LIN {X 0,Y 272.161,Z 198.873,A -85,B 0,C 180,E1 -18848.578,E2 -18848.578} C_VEL
LIN {X 0,Y 269.803,Z 194.303,A -85,B 0,C 180,E1 -18849.734,E2 -18849.734} C_VEL
LIN {X 0,Y 266.598,Z 188.645,A -85,B 0,C 180,E1 -18851.406,E2 -18851.406} C_VEL
LIN {X 0,Y 262.771,Z 182.274,A -85,B 0,C 180,E1 -18853.688,E2 -18853.688} C_VEL
LIN {X 0,Y 258.268,Z 175.293,A -85,B 0,C 180,E1 -18857.039,E2 -18857.039} C_VEL
LIN {X 0,Y 254.053,Z 169.261,A -85,B 0,C 180,E1 -18861.694,E2 -18861.694} C_VEL
LIN {X 0,Y 252.896,Z 167.097,A -85,B 0,C 180,E1 -18864.05,E2 -18864.05} C_VEL
LIN {X 0,Y 252.189,Z 165.744,A -85,B 0,C 180,E1 -18867.234,E2 -18867.234} C_VEL
LIN {X 0,Y 252.626,Z 165.739,A -85,B 0,C 180,E1 -18870.81,E2 -18870.81} C_VEL
LIN {X 0,Y 254.505,Z 167.542,A -85,B 0,C 180,E1 -18874.522,E2 -18874.522} C_VEL
LIN {X 0,Y 256.623,Z 169.192,A -85,B 0,C 180,E1 -18876.922,E2 -18876.922} C_VEL
LIN {X 0,Y 261.122,Z 174.199,A -85,B 0,C 180,E1 -18880.646,E2 -18880.646} C_VEL
LIN {X 0,Y 265.231,Z 179.251,A -85,B 0,C 180,E1 -18883.234,E2 -18883.234} C_VEL
LIN {X 0,Y 268.61,Z 183.835,A -85,B 0,C 180,E1 -18885.072,E2 -18885.072} C_VEL
LIN {X 0,Y 271.817,Z 188.374,A -85,B 0,C 180,E1 -18886.589,E2 -18886.589} C_VEL
LIN {X 0,Y 276.316,Z 195.238,A -85,B 0,C 180,E1 -18888.534,E2 -18888.534} C_VEL
LIN {X 0,Y 282.169,Z 206.406,A -85,B 0,C 180,E1 -18890.864,E2 -18890.864} C_VEL
LIN {X 0,Y 283.422,Z 209.263,A -85,B 0,C 180,E1 -18891.341,E2 -18891.341} C_VEL
LIN {X 0,Y 278.255,Z 265.436,A -85,B 0,C 180,E1 -18893.382,E2 -18893.382} C_VEL
LIN {X 0,Y 276.562,Z 278.897,A -85,B 0,C 180,E1 -18894.165,E2 -18894.165} C_VEL
LIN {X 0,Y 274.571,Z 290.757,A -85,B 0,C 180,E1 -18895.117,E2 -18895.117} C_VEL
LIN {X 0,Y 271.722,Z 303.647,A -85,B 0,C 180,E1 -18896.478,E2 -18896.478} C_VEL
LIN {X 0,Y 268.861,Z 314.419,A -85,B 0,C 180,E1 -18897.94,E2 -18897.94} C_VEL
LIN {X 0,Y 265.559,Z 325.122,A -85,B 0,C 180,E1 -18899.802,E2 -18899.802} C_VEL
LIN {X 0,Y 262.251,Z 334.733,A -85,B 0,C 180,E1 -18901.909,E2 -18901.909} C_VEL
LIN {X 0,Y 258.95,Z 343.17,A -85,B 0,C 180,E1 -18904.279,E2 -18904.279} C_VEL
LIN {X 0,Y 255.863,Z 350.386,A -85,B 0,C 180,E1 -18906.908,E2 -18906.908} C_VEL
LIN {X 0,Y 253.246,Z 355.852,A -85,B 0,C 180,E1 -18909.584,E2 -18909.584} C_VEL
LIN {X 0,Y 251.415,Z 359.437,A -85,B 0,C 180,E1 -18911.933,E2 -18911.933} C_VEL
LIN {X 0,Y 249.746,Z 362.315,A -85,B 0,C 180,E1 -18914.67,E2 -18914.67} C_VEL
LIN {X 0,Y 248.899,Z 363.505,A -85,B 0,C 180,E1 -18916.401,E2 -18916.401} C_VEL
LIN {X 0,Y 248.206,Z 364.182,A -85,B 0,C 180,E1 -18918.147,E2 -18918.147} C_VEL
LIN {X 0,Y 247.543,Z 364.385,A -85,B 0,C 180,E1 -18920.461,E2 -18920.461} C_VEL
LIN {X 0,Y 247.05,Z 363.363,A -85,B 0,C 180,E1 -18923.469,E2 -18923.469} C_VEL
LIN {X 0,Y 246.899,Z 362.091,A -85,B 0,C 180,E1 -18925.275,E2 -18925.275} C_VEL
LIN {X 0,Y 247.04,Z 358.996,A -85,B 0,C 180,E1 -18928.125,E2 -18928.125} C_VEL
LIN {X 0,Y 247.409,Z 354.863,A -85,B 0,C 180,E1 -18930.751,E2 -18930.751} C_VEL
LIN {X 0,Y 247.931,Z 348.96,A -85,B 0,C 180,E1 -18933.556,E2 -18933.556} C_VEL
LIN {X 0,Y 248.602,Z 342.47,A -85,B 0,C 180,E1 -18935.968,E2 -18935.968} C_VEL
LIN {X 0,Y 249.5,Z 334.669,A -85,B 0,C 180,E1 -18938.294,E2 -18938.294} C_VEL
LIN {X 0,Y 250.624,Z 325.418,A -85,B 0,C 180,E1 -18940.519,E2 -18940.519} C_VEL
LIN {X 0,Y 251.866,Z 314.797,A -85,B 0,C 180,E1 -18942.583,E2 -18942.583} C_VEL
LIN {X 0,Y 253.111,Z 304.125,A -85,B 0,C 180,E1 -18944.236,E2 -18944.236} C_VEL
LIN {X 0,Y 254.279,Z 291.49,A -85,B 0,C 180,E1 -18945.797,E2 -18945.797} C_VEL
LIN {X 0,Y 255.46,Z 277.915,A -85,B 0,C 180,E1 -18947.043,E2 -18947.043} C_VEL
LIN {X 0,Y 256.185,Z 264.7,A -85,B 0,C 180,E1 -18947.927,E2 -18947.927} C_VEL
LIN {X 0,Y 256.929,Z 247.419,A -85,B 0,C 180,E1 -18948.64,E2 -18948.64} C_VEL
LIN {X 0,Y 259.313,Z 186.757,A -85,B 0,C 180,E1 -18950.805,E2 -18950.805} C_VEL
LIN {X 0,Y 254.059,Z 171.401,A -85,B 0,C 180,E1 -18951.759,E2 -18951.759} C_VEL
LIN {X 0,Y 249.108,Z 157.454,A -85,B 0,C 180,E1 -18952.7,E2 -18952.7} C_VEL
LIN {X 0,Y 249.056,Z 157.463,A -85,B 0,C 180,E1 -18955.641,E2 -18955.641} C_VEL
LIN {X 0,Y 249.052,Z 157.465,A -85,B 0,C 180,E1 -18959.472,E2 -18959.472} C_VEL
LIN {X 0,Y 249.074,Z 157.462,A -85,B 0,C 180,E1 -18963.162,E2 -18963.162} C_VEL
LIN {X 0,Y 249.078,Z 157.458,A -85,B 0,C 180,E1 -18966.732,E2 -18966.732} C_VEL
LIN {X 0,Y 249.092,Z 157.454,A -85,B 0,C 180,E1 -18970.209,E2 -18970.209} C_VEL
LIN {X 0,Y 249.194,Z 157.443,A -85,B 0,C 180,E1 -18973.618,E2 -18973.618} C_VEL
LIN {X 0,Y 249.25,Z 157.436,A -85,B 0,C 180,E1 -18978.616,E2 -18978.616} C_VEL
LIN {X 0,Y 249.478,Z 157.406,A -85,B 0,C 180,E1 -18981.902,E2 -18981.902} C_VEL
LIN {X 0,Y 249.435,Z 157.414,A -85,B 0,C 180,E1 -18986.769,E2 -18986.769} C_VEL
LIN {X 0,Y 249.727,Z 157.376,A -85,B 0,C 180,E1 -18989.999,E2 -18989.999} C_VEL
LIN {X 0,Y 249.434,Z 157.412,A -85,B 0,C 180,E1 -18993.23,E2 -18993.23} C_VEL
LIN {X 0,Y 249.478,Z 157.408,A -85,B 0,C 180,E1 -18998.097,E2 -18998.097} C_VEL
LIN {X 0,Y 249.251,Z 157.433,A -85,B 0,C 180,E1 -19001.383,E2 -19001.383} C_VEL
LIN {X 0,Y 249.24,Z 157.44,A -85,B 0,C 180,E1 -19006.378,E2 -19006.378} C_VEL
LIN {X 0,Y 249.081,Z 157.455,A -85,B 0,C 180,E1 -19011.518,E2 -19011.518} C_VEL
LIN {X 0,Y 249.115,Z 157.452,A -85,B 0,C 180,E1 -19015.475,E2 -19015.475} C_VEL
LIN {X 0,Y 249.084,Z 157.455,A -85,B 0,C 180,E1 -19018.994,E2 -19018.994} C_VEL
LIN {X 0,Y 249.033,Z 157.464,A -85,B 0,C 180,E1 -19022.425,E2 -19022.425} C_VEL
LIN {X 0,Y 249.072,Z 157.458,A -85,B 0,C 180,E1 -19026.337,E2 -19026.337} C_VEL
LIN {X 0,Y 249.074,Z 157.458,A -85,B 0,C 180,E1 -19030.464,E2 -19030.464} C_VEL
LIN {X 0,Y 249.019,Z 157.462,A -85,B 0,C 180,E1 -19034.875,E2 -19034.875} C_VEL
LIN {X 0,Y 249.049,Z 157.461,A -85,B 0,C 180,E1 -19037.371,E2 -19037.371} C_VEL
LIN {X 0,Y 249.048,Z 157.463,A -85,B 0,C 180,E1 -19041.624,E2 -19041.624} C_VEL
LIN {X 0,Y 249.059,Z 157.463,A -85,B 0,C 180,E1 -19045.643,E2 -19045.643} C_VEL
LIN {X 0,Y 249.049,Z 157.463,A -85,B 0,C 180,E1 -19049.473,E2 -19049.473} C_VEL
LIN {X 0,Y 249.072,Z 157.459,A -85,B 0,C 180,E1 -19053.163,E2 -19053.163} C_VEL
LIN {X 0,Y 249.077,Z 157.457,A -85,B 0,C 180,E1 -19056.733,E2 -19056.733} C_VEL
LIN {X 0,Y 249.108,Z 157.451,A -85,B 0,C 180,E1 -19060.212,E2 -19060.212} C_VEL
LIN {X 0,Y 249.239,Z 157.438,A -85,B 0,C 180,E1 -19063.622,E2 -19063.622} C_VEL
LIN {X 0,Y 249.251,Z 157.434,A -85,B 0,C 180,E1 -19068.617,E2 -19068.617} C_VEL
LIN {X 0,Y 249.477,Z 157.407,A -85,B 0,C 180,E1 -19071.903,E2 -19071.903} C_VEL
LIN {X 0,Y 249.434,Z 157.413,A -85,B 0,C 180,E1 -19076.77,E2 -19076.77} C_VEL
LIN {X 0,Y 249.727,Z 157.376,A -85,B 0,C 180,E1 -19080.001,E2 -19080.001} C_VEL
LIN {X 0,Y 249.435,Z 157.411,A -85,B 0,C 180,E1 -19083.231,E2 -19083.231} C_VEL
LIN {X 0,Y 249.483,Z 157.407,A -85,B 0,C 180,E1 -19088.098,E2 -19088.098} C_VEL
LIN {X 0,Y 249.252,Z 157.433,A -85,B 0,C 180,E1 -19091.384,E2 -19091.384} C_VEL
LIN {X 0,Y 249.206,Z 157.441,A -85,B 0,C 180,E1 -19095.849,E2 -19095.849} C_VEL
LIN {X 0,Y 248.917,Z 157.479,A -85,B 0,C 180,E1 -19096.751,E2 -19096.751} C_VEL
LIN {X 0,Y 247.56,Z 157.65,A -85,B 0,C 180,E1 -19098.081,E2 -19098.081} C_VEL
LIN {X 0,Y 243.133,Z 158.197,A -85,B 0,C 180,E1 -19101.182,E2 -19101.182} C_VEL
LIN {X 0,Y 242.07,Z 158.332,A -85,B 0,C 180,E1 -19102.572,E2 -19102.572} C_VEL
LIN {X 0,Y 241.992,Z 158.337,A -85,B 0,C 180,E1 -19103.044,E2 -19103.044} C_VEL
LIN {X 0,Y 242.066,Z 158.331,A -85,B 0,C 180,E1 -19105.839,E2 -19105.839} C_VEL
LIN {X 0,Y 242.03,Z 158.333,A -85,B 0,C 180,E1 -19109.581,E2 -19109.581} C_VEL
LIN {X 0,Y 241.991,Z 158.34,A -85,B 0,C 180,E1 -19113.492,E2 -19113.492} C_VEL
LIN {X 0,Y 242.011,Z 158.335,A -85,B 0,C 180,E1 -19117.579,E2 -19117.579} C_VEL
LIN {X 0,Y 241.954,Z 158.348,A -85,B 0,C 180,E1 -19121.92,E2 -19121.92} C_VEL
LIN {X 0,Y 241.935,Z 158.347,A -85,B 0,C 180,E1 -19126.572,E2 -19126.572} C_VEL
LIN {X 0,Y 241.957,Z 158.345,A -85,B 0,C 180,E1 -19130.282,E2 -19130.282} C_VEL
LIN {X 0,Y 242.087,Z 158.358,A -85,B 0,C 180,E1 -19134.698,E2 -19134.698} C_VEL
LIN {X 0,Y 244.791,Z 171.849,A -85,B 0,C 180,E1 -19139.464,E2 -19139.464} C_VEL
LIN {X 0,Y 246.244,Z 179.046,A -85,B 0,C 180,E1 -19141.867,E2 -19141.867} C_VEL
LIN {X 0,Y 251.436,Z 230.762,A -85,B 0,C 180,E1 -19144.295,E2 -19144.295} C_VEL
LIN {X 0,Y 249.178,Z 289.171,A -85,B 0,C 180,E1 -19146.523,E2 -19146.523} C_VEL
LIN {X 0,Y 248.278,Z 301.999,A -85,B 0,C 180,E1 -19147.315,E2 -19147.315} C_VEL
LIN {X 0,Y 247.106,Z 313.577,A -85,B 0,C 180,E1 -19148.301,E2 -19148.301} C_VEL
LIN {X 0,Y 245.772,Z 325.986,A -85,B 0,C 180,E1 -19149.714,E2 -19149.714} C_VEL
LIN {X 0,Y 244.389,Z 337.207,A -85,B 0,C 180,E1 -19151.342,E2 -19151.342} C_VEL
LIN {X 0,Y 243.042,Z 347.408,A -85,B 0,C 180,E1 -19153.193,E2 -19153.193} C_VEL
LIN {X 0,Y 242.034,Z 356.689,A -85,B 0,C 180,E1 -19155.282,E2 -19155.282} C_VEL
LIN {X 0,Y 241.063,Z 365.717,A -85,B 0,C 180,E1 -19157.798,E2 -19157.798} C_VEL
LIN {X 0,Y 240.491,Z 372.88,A -85,B 0,C 180,E1 -19160.327,E2 -19160.327} C_VEL
LIN {X 0,Y 240.242,Z 379.387,A -85,B 0,C 180,E1 -19163.281,E2 -19163.281} C_VEL
LIN {X 0,Y 240.242,Z 383.565,A -85,B 0,C 180,E1 -19165.807,E2 -19165.807} C_VEL
LIN {X 0,Y 240.167,Z 386.556,A -85,B 0,C 180,E1 -19168.324,E2 -19168.324} C_VEL
LIN {X 0,Y 240.34,Z 387.982,A -85,B 0,C 180,E1 -19170.001,E2 -19170.001} C_VEL
LIN {X 0,Y 240.01,Z 389.407,A -85,B 0,C 180,E1 -19173.358,E2 -19173.358} C_VEL
LIN {X 0,Y 239.853,Z 389.5,A -85,B 0,C 180,E1 -19175.044,E2 -19175.044} C_VEL
LIN {X 0,Y 239.896,Z 389.18,A -85,B 0,C 180,E1 -19176.73,E2 -19176.73} C_VEL
LIN {X 0,Y 240.5,Z 387.299,A -85,B 0,C 180,E1 -19180.099,E2 -19180.099} C_VEL
LIN {X 0,Y 241.037,Z 385.763,A -85,B 0,C 180,E1 -19181.778,E2 -19181.778} C_VEL
LIN {X 0,Y 242.247,Z 382.634,A -85,B 0,C 180,E1 -19184.277,E2 -19184.277} C_VEL
LIN {X 0,Y 244.074,Z 378.522,A -85,B 0,C 180,E1 -19186.736,E2 -19186.736} C_VEL
LIN {X 0,Y 246.158,Z 373.316,A -85,B 0,C 180,E1 -19189.168,E2 -19189.168} C_VEL
LIN {X 0,Y 248.789,Z 366.863,A -85,B 0,C 180,E1 -19191.546,E2 -19191.546} C_VEL
LIN {X 0,Y 252.077,Z 358.919,A -85,B 0,C 180,E1 -19193.846,E2 -19193.846} C_VEL
LIN {X 0,Y 255.101,Z 350.996,A -85,B 0,C 180,E1 -19195.717,E2 -19195.717} C_VEL
LIN {X 0,Y 258.965,Z 340.381,A -85,B 0,C 180,E1 -19197.695,E2 -19197.695} C_VEL
LIN {X 0,Y 262.272,Z 329.818,A -85,B 0,C 180,E1 -19199.278,E2 -19199.278} C_VEL
LIN {X 0,Y 265.545,Z 318.133,A -85,B 0,C 180,E1 -19200.63,E2 -19200.63} C_VEL
LIN {X 0,Y 268.928,Z 304.154,A -85,B 0,C 180,E1 -19201.842,E2 -19201.842} C_VEL
LIN {X 0,Y 271.411,Z 290.859,A -85,B 0,C 180,E1 -19202.666,E2 -19202.666} C_VEL
LIN {X 0,Y 273.13,Z 276.909,A -85,B 0,C 180,E1 -19203.288,E2 -19203.288} C_VEL
LIN {X 0,Y 276.662,Z 237.361,A -85,B 0,C 180,E1 -19204.745,E2 -19204.745} C_VEL
LIN {X 0,Y 275.715,Z 223.84,A -85,B 0,C 180,E1 -19205.824,E2 -19205.824} C_VEL
LIN {X 0,Y 275.099,Z 218.549,A -85,B 0,C 180,E1 -19206.339,E2 -19206.339} C_VEL
LIN {X 0,Y 271.495,Z 209.724,A -85,B 0,C 180,E1 -19208.005,E2 -19208.005} C_VEL
LIN {X 0,Y 267.297,Z 200.762,A -85,B 0,C 180,E1 -19210.135,E2 -19210.135} C_VEL
LIN {X 0,Y 263.888,Z 194.57,A -85,B 0,C 180,E1 -19212.024,E2 -19212.024} C_VEL
LIN {X 0,Y 260.503,Z 188.645,A -85,B 0,C 180,E1 -19214.173,E2 -19214.173} C_VEL
LIN {X 0,Y 256.366,Z 181.862,A -85,B 0,C 180,E1 -19217.45,E2 -19217.45} C_VEL
LIN {X 0,Y 252.367,Z 175.801,A -85,B 0,C 180,E1 -19222.217,E2 -19222.217} C_VEL
LIN {X 0,Y 251.349,Z 173.787,A -85,B 0,C 180,E1 -19224.568,E2 -19224.568} C_VEL
LIN {X 0,Y 250.805,Z 172.582,A -85,B 0,C 180,E1 -19227.831,E2 -19227.831} C_VEL
LIN {X 0,Y 251.371,Z 172.83,A -85,B 0,C 180,E1 -19231.136,E2 -19231.136} C_VEL
LIN {X 0,Y 253.916,Z 175.089,A -85,B 0,C 180,E1 -19235.469,E2 -19235.469} C_VEL
LIN {X 0,Y 255.04,Z 176.102,A -85,B 0,C 180,E1 -19236.744,E2 -19236.744} C_VEL
LIN {X 0,Y 259.027,Z 180.69,A -85,B 0,C 180,E1 -19240.204,E2 -19240.204} C_VEL
LIN {X 0,Y 262.925,Z 185.673,A -85,B 0,C 180,E1 -19242.798,E2 -19242.798} C_VEL
LIN {X 0,Y 266.299,Z 190.371,A -85,B 0,C 180,E1 -19244.697,E2 -19244.697} C_VEL
LIN {X 0,Y 270.776,Z 197.051,A -85,B 0,C 180,E1 -19246.892,E2 -19246.892} C_VEL
LIN {X 0,Y 274.226,Z 203.049,A -85,B 0,C 180,E1 -19248.441,E2 -19248.441} C_VEL
LIN {X 0,Y 278.658,Z 212.019,A -85,B 0,C 180,E1 -19250.306,E2 -19250.306} C_VEL
LIN {X 0,Y 273.522,Z 265.759,A -85,B 0,C 180,E1 -19252.285,E2 -19252.285} C_VEL
LIN {X 0,Y 271.809,Z 278.655,A -85,B 0,C 180,E1 -19253.038,E2 -19253.038} C_VEL
LIN {X 0,Y 269.661,Z 290.779,A -85,B 0,C 180,E1 -19254.016,E2 -19254.016} C_VEL
LIN {X 0,Y 266.869,Z 302.828,A -85,B 0,C 180,E1 -19255.289,E2 -19255.289} C_VEL
LIN {X 0,Y 263.827,Z 313.801,A -85,B 0,C 180,E1 -19256.754,E2 -19256.754} C_VEL
LIN {X 0,Y 260.656,Z 323.839,A -85,B 0,C 180,E1 -19258.454,E2 -19258.454} C_VEL
LIN {X 0,Y 257.324,Z 332.949,A -85,B 0,C 180,E1 -19260.391,E2 -19260.391} C_VEL
LIN {X 0,Y 253.79,Z 341.769,A -85,B 0,C 180,E1 -19262.776,E2 -19262.776} C_VEL
LIN {X 0,Y 250.61,Z 348.832,A -85,B 0,C 180,E1 -19265.229,E2 -19265.229} C_VEL
LIN {X 0,Y 248.095,Z 353.926,A -85,B 0,C 180,E1 -19267.484,E2 -19267.484} C_VEL
LIN {X 0,Y 245.868,Z 358.084,A -85,B 0,C 180,E1 -19269.875,E2 -19269.875} C_VEL
LIN {X 0,Y 244.28,Z 360.854,A -85,B 0,C 180,E1 -19271.986,E2 -19271.986} C_VEL
LIN {X 0,Y 242.399,Z 363.55,A -85,B 0,C 180,E1 -19275.125,E2 -19275.125} C_VEL
LIN {X 0,Y 241.591,Z 364.425,A -85,B 0,C 180,E1 -19276.911,E2 -19276.911} C_VEL
LIN {X 0,Y 240.912,Z 364.831,A -85,B 0,C 180,E1 -19278.717,E2 -19278.717} C_VEL
LIN {X 0,Y 240.405,Z 364.695,A -85,B 0,C 180,E1 -19280.692,E2 -19280.692} C_VEL
LIN {X 0,Y 240.068,Z 364.163,A -85,B 0,C 180,E1 -19282.369,E2 -19282.369} C_VEL
LIN {X 0,Y 239.846,Z 362.691,A -85,B 0,C 180,E1 -19284.718,E2 -19284.718} C_VEL
LIN {X 0,Y 239.915,Z 359.335,A -85,B 0,C 180,E1 -19287.949,E2 -19287.949} C_VEL
LIN {X 0,Y 240.306,Z 354.927,A -85,B 0,C 180,E1 -19290.783,E2 -19290.783} C_VEL
LIN {X 0,Y 240.873,Z 348.928,A -85,B 0,C 180,E1 -19293.666,E2 -19293.666} C_VEL
LIN {X 0,Y 241.548,Z 342.465,A -85,B 0,C 180,E1 -19296.099,E2 -19296.099} C_VEL
LIN {X 0,Y 242.477,Z 334.497,A -85,B 0,C 180,E1 -19298.502,E2 -19298.502} C_VEL
LIN {X 0,Y 243.618,Z 325.33,A -85,B 0,C 180,E1 -19300.744,E2 -19300.744} C_VEL
LIN {X 0,Y 244.706,Z 315.837,A -85,B 0,C 180,E1 -19302.643,E2 -19302.643} C_VEL
LIN {X 0,Y 246.029,Z 304.743,A -85,B 0,C 180,E1 -19304.426,E2 -19304.426} C_VEL
LIN {X 0,Y 247.246,Z 292.317,A -85,B 0,C 180,E1 -19306.013,E2 -19306.013} C_VEL
LIN {X 0,Y 248.356,Z 279.879,A -85,B 0,C 180,E1 -19307.222,E2 -19307.222} C_VEL
LIN {X 0,Y 249.236,Z 265.509,A -85,B 0,C 180,E1 -19308.238,E2 -19308.238} C_VEL
LIN {X 0,Y 249.988,Z 249.032,A -85,B 0,C 180,E1 -19308.957,E2 -19308.957} C_VEL
LIN {X 0,Y 252.492,Z 188.132,A -85,B 0,C 180,E1 -19311.209,E2 -19311.209} C_VEL
LIN {X 0,Y 245.433,Z 167.869,A -85,B 0,C 180,E1 -19312.519,E2 -19312.519} C_VEL
LIN {X 0,Y 242.051,Z 158.335,A -85,B 0,C 180,E1 -19313.182,E2 -19313.182} C_VEL
LIN {X 0,Y 241.993,Z 158.343,A -85,B 0,C 180,E1 -19317.374,E2 -19317.374} C_VEL
LIN {X 0,Y 242.037,Z 158.336,A -85,B 0,C 180,E1 -19320.586,E2 -19320.586} C_VEL
LIN {X 0,Y 242.067,Z 158.331,A -85,B 0,C 180,E1 -19324.182,E2 -19324.182} C_VEL
LIN {X 0,Y 242.051,Z 158.332,A -85,B 0,C 180,E1 -19328.297,E2 -19328.297} C_VEL
LIN {X 0,Y 242.114,Z 158.327,A -85,B 0,C 180,E1 -19333.315,E2 -19333.315} C_VEL
LIN {X 0,Y 242.182,Z 158.315,A -85,B 0,C 180,E1 -19338.279,E2 -19338.279} C_VEL
LIN {X 0,Y 242.425,Z 158.286,A -85,B 0,C 180,E1 -19341.665,E2 -19341.665} C_VEL
LIN {X 0,Y 242.258,Z 158.308,A -85,B 0,C 180,E1 -19345.007,E2 -19345.007} C_VEL
LIN {X 0,Y 242.635,Z 158.26,A -85,B 0,C 180,E1 -19348.34,E2 -19348.34} C_VEL
LIN {X 0,Y 242.635,Z 158.258,A -85,B 0,C 180,E1 -19351.659,E2 -19351.659} C_VEL
LIN {X 0,Y 242.43,Z 158.289,A -85,B 0,C 180,E1 -19356.658,E2 -19356.658} C_VEL
LIN {X 0,Y 242.312,Z 158.299,A -85,B 0,C 180,E1 -19360.021,E2 -19360.021} C_VEL
LIN {X 0,Y 242.165,Z 158.318,A -85,B 0,C 180,E1 -19365.14,E2 -19365.14} C_VEL
LIN {X 0,Y 242.07,Z 158.33,A -85,B 0,C 180,E1 -19368.624,E2 -19368.624} C_VEL
LIN {X 0,Y 242.004,Z 158.34,A -85,B 0,C 180,E1 -19372.18,E2 -19372.18} C_VEL
LIN {X 0,Y 242.064,Z 158.331,A -85,B 0,C 180,E1 -19375.838,E2 -19375.838} C_VEL
LIN {X 0,Y 242.029,Z 158.334,A -85,B 0,C 180,E1 -19379.58,E2 -19379.58} C_VEL
LIN {X 0,Y 241.989,Z 158.34,A -85,B 0,C 180,E1 -19383.491,E2 -19383.491} C_VEL
LIN {X 0,Y 242.01,Z 158.337,A -85,B 0,C 180,E1 -19387.577,E2 -19387.577} C_VEL
LIN {X 0,Y 241.982,Z 158.344,A -85,B 0,C 180,E1 -19391.912,E2 -19391.912} C_VEL
LIN {X 0,Y 241.982,Z 158.34,A -85,B 0,C 180,E1 -19396.558,E2 -19396.558} C_VEL
LIN {X 0,Y 241.985,Z 158.34,A -85,B 0,C 180,E1 -19400.287,E2 -19400.287} C_VEL
LIN {X 0,Y 242.033,Z 158.333,A -85,B 0,C 180,E1 -19404.498,E2 -19404.498} C_VEL
LIN {X 0,Y 241.973,Z 158.341,A -85,B 0,C 180,E1 -19408.48,E2 -19408.48} C_VEL
LIN {X 0,Y 242.006,Z 158.336,A -85,B 0,C 180,E1 -19412.313,E2 -19412.313} C_VEL
LIN {X 0,Y 242.055,Z 158.332,A -85,B 0,C 180,E1 -19416.016,E2 -19416.016} C_VEL
LIN {X 0,Y 242.035,Z 158.335,A -85,B 0,C 180,E1 -19419.608,E2 -19419.608} C_VEL
LIN {X 0,Y 242.161,Z 158.322,A -85,B 0,C 180,E1 -19423.279,E2 -19423.279} C_VEL
LIN {X 0,Y 242.184,Z 158.313,A -85,B 0,C 180,E1 -19428.28,E2 -19428.28} C_VEL
LIN {X 0,Y 242.424,Z 158.286,A -85,B 0,C 180,E1 -19431.666,E2 -19431.666} C_VEL
LIN {X 0,Y 242.258,Z 158.308,A -85,B 0,C 180,E1 -19435.008,E2 -19435.008} C_VEL
LIN {X 0,Y 242.635,Z 158.259,A -85,B 0,C 180,E1 -19438.341,E2 -19438.341} C_VEL
LIN {X 0,Y 242.635,Z 158.259,A -85,B 0,C 180,E1 -19441.66,E2 -19441.66} C_VEL
LIN {X 0,Y 242.433,Z 158.287,A -85,B 0,C 180,E1 -19446.659,E2 -19446.659} C_VEL
LIN {X 0,Y 242.344,Z 158.296,A -85,B 0,C 180,E1 -19450.021,E2 -19450.021} C_VEL
LIN {X 0,Y 242.166,Z 158.318,A -85,B 0,C 180,E1 -19455.141,E2 -19455.141} C_VEL
LIN {X 0,Y 242.072,Z 158.331,A -85,B 0,C 180,E1 -19458.625,E2 -19458.625} C_VEL
LIN {X 0,Y 241.992,Z 158.337,A -85,B 0,C 180,E1 -19463.044,E2 -19463.044} C_VEL
LIN {X 0,Y 241.352,Z 158.423,A -85,B 0,C 180,E1 -19464.432,E2 -19464.432} C_VEL
LIN {X 0,Y 238.523,Z 158.772,A -85,B 0,C 180,E1 -19466.696,E2 -19466.696} C_VEL
LIN {X 0,Y 236.093,Z 159.074,A -85,B 0,C 180,E1 -19468.541,E2 -19468.541} C_VEL
LIN {X 0,Y 235.031,Z 159.206,A -85,B 0,C 180,E1 -19469.972,E2 -19469.972} C_VEL
LIN {X 0,Y 234.935,Z 159.219,A -85,B 0,C 180,E1 -19470.458,E2 -19470.458} C_VEL
LIN {X 0,Y 234.96,Z 159.216,A -85,B 0,C 180,E1 -19474.634,E2 -19474.634} C_VEL
LIN {X 0,Y 234.942,Z 159.217,A -85,B 0,C 180,E1 -19478.945,E2 -19478.945} C_VEL
LIN {X 0,Y 234.921,Z 159.221,A -85,B 0,C 180,E1 -19483.479,E2 -19483.479} C_VEL
LIN {X 0,Y 234.888,Z 159.225,A -85,B 0,C 180,E1 -19486.515,E2 -19486.515} C_VEL
LIN {X 0,Y 234.919,Z 159.221,A -85,B 0,C 180,E1 -19491.08,E2 -19491.08} C_VEL
LIN {X 0,Y 235.058,Z 159.348,A -85,B 0,C 180,E1 -19494.418,E2 -19494.418} C_VEL
LIN {X 0,Y 237.284,Z 170.542,A -85,B 0,C 180,E1 -19498.505,E2 -19498.505} C_VEL
LIN {X 0,Y 238.974,Z 178.656,A -85,B 0,C 180,E1 -19501.322,E2 -19501.322} C_VEL
LIN {X 0,Y 239.927,Z 182.771,A -85,B 0,C 180,E1 -19501.567,E2 -19501.567} C_VEL
LIN {X 0,Y 244.528,Z 231.857,A -85,B 0,C 180,E1 -19503.924,E2 -19503.924} C_VEL
LIN {X 0,Y 242.294,Z 288.298,A -85,B 0,C 180,E1 -19506.155,E2 -19506.155} C_VEL
LIN {X 0,Y 241.354,Z 301.216,A -85,B 0,C 180,E1 -19506.966,E2 -19506.966} C_VEL
LIN {X 0,Y 240.074,Z 313.903,A -85,B 0,C 180,E1 -19508.085,E2 -19508.085} C_VEL
LIN {X 0,Y 238.715,Z 326.148,A -85,B 0,C 180,E1 -19509.537,E2 -19509.537} C_VEL
LIN {X 0,Y 237.253,Z 337.811,A -85,B 0,C 180,E1 -19511.303,E2 -19511.303} C_VEL
LIN {X 0,Y 235.955,Z 347.372,A -85,B 0,C 180,E1 -19513.118,E2 -19513.118} C_VEL
LIN {X 0,Y 234.942,Z 356.6,A -85,B 0,C 180,E1 -19515.271,E2 -19515.271} C_VEL
LIN {X 0,Y 233.976,Z 365.573,A -85,B 0,C 180,E1 -19517.863,E2 -19517.863} C_VEL
LIN {X 0,Y 233.417,Z 372.681,A -85,B 0,C 180,E1 -19520.469,E2 -19520.469} C_VEL
LIN {X 0,Y 233.181,Z 378.316,A -85,B 0,C 180,E1 -19523.076,E2 -19523.076} C_VEL
LIN {X 0,Y 233.188,Z 382.654,A -85,B 0,C 180,E1 -19525.68,E2 -19525.68} C_VEL
LIN {X 0,Y 233.097,Z 385.784,A -85,B 0,C 180,E1 -19528.273,E2 -19528.273} C_VEL
LIN {X 0,Y 233.262,Z 387.301,A -85,B 0,C 180,E1 -19530.001,E2 -19530.001} C_VEL
LIN {X 0,Y 232.969,Z 388.309,A -85,B 0,C 180,E1 -19531.729,E2 -19531.729} C_VEL
LIN {X 0,Y 232.937,Z 388.888,A -85,B 0,C 180,E1 -19533.46,E2 -19533.46} C_VEL
LIN {X 0,Y 232.846,Z 388.825,A -85,B 0,C 180,E1 -19536.935,E2 -19536.935} C_VEL
LIN {X 0,Y 233.084,Z 388.195,A -85,B 0,C 180,E1 -19538.672,E2 -19538.672} C_VEL
LIN {X 0,Y 234.042,Z 385.677,A -85,B 0,C 180,E1 -19542.135,E2 -19542.135} C_VEL
LIN {X 0,Y 235.358,Z 382.732,A -85,B 0,C 180,E1 -19544.704,E2 -19544.704} C_VEL
LIN {X 0,Y 237.278,Z 378.785,A -85,B 0,C 180,E1 -19547.23,E2 -19547.23} C_VEL
LIN {X 0,Y 239.808,Z 372.863,A -85,B 0,C 180,E1 -19550.113,E2 -19550.113} C_VEL
LIN {X 0,Y 242.783,Z 366.383,A -85,B 0,C 180,E1 -19552.555,E2 -19552.555} C_VEL
LIN {X 0,Y 246.306,Z 358.502,A -85,B 0,C 180,E1 -19554.89,E2 -19554.89} C_VEL
LIN {X 0,Y 249.51,Z 350.573,A -85,B 0,C 180,E1 -19556.788,E2 -19556.788} C_VEL
LIN {X 0,Y 253.59,Z 339.938,A -85,B 0,C 180,E1 -19558.786,E2 -19558.786} C_VEL
LIN {X 0,Y 257.104,Z 329.488,A -85,B 0,C 180,E1 -19560.379,E2 -19560.379} C_VEL
LIN {X 0,Y 260.083,Z 319.603,A -85,B 0,C 180,E1 -19561.572,E2 -19561.572} C_VEL
LIN {X 0,Y 263.562,Z 306.217,A -85,B 0,C 180,E1 -19562.796,E2 -19562.796} C_VEL
LIN {X 0,Y 266.265,Z 293.281,A -85,B 0,C 180,E1 -19563.662,E2 -19563.662} C_VEL
LIN {X 0,Y 268.276,Z 279.041,A -85,B 0,C 180,E1 -19564.337,E2 -19564.337} C_VEL
LIN {X 0,Y 272.163,Z 238.757,A -85,B 0,C 180,E1 -19565.854,E2 -19565.854} C_VEL
LIN {X 0,Y 271.147,Z 222.952,A -85,B 0,C 180,E1 -19567.197,E2 -19567.197} C_VEL
LIN {X 0,Y 268.34,Z 215.423,A -85,B 0,C 180,E1 -19568.626,E2 -19568.626} C_VEL
LIN {X 0,Y 264.254,Z 206.386,A -85,B 0,C 180,E1 -19570.815,E2 -19570.815} C_VEL
LIN {X 0,Y 261.112,Z 200.322,A -85,B 0,C 180,E1 -19572.712,E2 -19572.712} C_VEL
LIN {X 0,Y 258.062,Z 194.689,A -85,B 0,C 180,E1 -19574.821,E2 -19574.821} C_VEL
LIN {X 0,Y 254.394,Z 188.377,A -85,B 0,C 180,E1 -19577.936,E2 -19577.936} C_VEL
LIN {X 0,Y 250.788,Z 182.536,A -85,B 0,C 180,E1 -19582.571,E2 -19582.571} C_VEL
LIN {X 0,Y 249.96,Z 180.766,A -85,B 0,C 180,E1 -19584.626,E2 -19584.626} C_VEL
LIN {X 0,Y 249.46,Z 179.574,A -85,B 0,C 180,E1 -19587.693,E2 -19587.693} C_VEL
LIN {X 0,Y 249.948,Z 179.744,A -85,B 0,C 180,E1 -19590.957,E2 -19590.957} C_VEL
LIN {X 0,Y 252.416,Z 181.968,A -85,B 0,C 180,E1 -19595.313,E2 -19595.313} C_VEL
LIN {X 0,Y 253.64,Z 183.312,A -85,B 0,C 180,E1 -19596.77,E2 -19596.77} C_VEL
LIN {X 0,Y 257.047,Z 187.313,A -85,B 0,C 180,E1 -19599.829,E2 -19599.829} C_VEL
LIN {X 0,Y 260.559,Z 191.969,A -85,B 0,C 180,E1 -19602.292,E2 -19602.292} C_VEL
LIN {X 0,Y 263.976,Z 196.926,A -85,B 0,C 180,E1 -19604.313,E2 -19604.313} C_VEL
LIN {X 0,Y 267.803,Z 202.871,A -85,B 0,C 180,E1 -19606.297,E2 -19606.297} C_VEL
LIN {X 0,Y 270.934,Z 208.614,A -85,B 0,C 180,E1 -19607.817,E2 -19607.817} C_VEL
LIN {X 0,Y 274.094,Z 215.196,A -85,B 0,C 180,E1 -19609.222,E2 -19609.222} C_VEL
LIN {X 0,Y 268.858,Z 266.459,A -85,B 0,C 180,E1 -19611.165,E2 -19611.165} C_VEL
LIN {X 0,Y 266.975,Z 279.78,A -85,B 0,C 180,E1 -19611.96,E2 -19611.96} C_VEL
LIN {X 0,Y 264.705,Z 291.793,A -85,B 0,C 180,E1 -19612.946,E2 -19612.946} C_VEL
LIN {X 0,Y 261.832,Z 303.592,A -85,B 0,C 180,E1 -19614.215,E2 -19614.215} C_VEL
LIN {X 0,Y 258.568,Z 314.589,A -85,B 0,C 180,E1 -19615.713,E2 -19615.713} C_VEL
LIN {X 0,Y 254.855,Z 325.38,A -85,B 0,C 180,E1 -19617.61,E2 -19617.61} C_VEL
LIN {X 0,Y 251.006,Z 335.278,A -85,B 0,C 180,E1 -19619.825,E2 -19619.825} C_VEL
LIN {X 0,Y 247.736,Z 342.788,A -85,B 0,C 180,E1 -19621.951,E2 -19621.951} C_VEL
LIN {X 0,Y 244.25,Z 349.91,A -85,B 0,C 180,E1 -19624.538,E2 -19624.538} C_VEL
LIN {X 0,Y 240.979,Z 355.951,A -85,B 0,C 180,E1 -19627.434,E2 -19627.434} C_VEL
LIN {X 0,Y 238.498,Z 360.099,A -85,B 0,C 180,E1 -19630.183,E2 -19630.183} C_VEL
LIN {X 0,Y 237.139,Z 362.139,A -85,B 0,C 180,E1 -19632.036,E2 -19632.036} C_VEL
LIN {X 0,Y 236.056,Z 363.596,A -85,B 0,C 180,E1 -19633.779,E2 -19633.779} C_VEL
LIN {X 0,Y 234.625,Z 364.978,A -85,B 0,C 180,E1 -19636.556,E2 -19636.556} C_VEL
LIN {X 0,Y 233.625,Z 365.283,A -85,B 0,C 180,E1 -19639.323,E2 -19639.323} C_VEL
LIN {X 0,Y 233.187,Z 364.866,A -85,B 0,C 180,E1 -19641.202,E2 -19641.202} C_VEL
LIN {X 0,Y 232.865,Z 363.975,A -85,B 0,C 180,E1 -19643.1,E2 -19643.1} C_VEL
LIN {X 0,Y 232.744,Z 362.538,A -85,B 0,C 180,E1 -19645.056,E2 -19645.056} C_VEL
LIN {X 0,Y 232.813,Z 359.444,A -85,B 0,C 180,E1 -19647.898,E2 -19647.898} C_VEL
LIN {X 0,Y 233.205,Z 354.952,A -85,B 0,C 180,E1 -19650.818,E2 -19650.818} C_VEL
LIN {X 0,Y 233.79,Z 348.864,A -85,B 0,C 180,E1 -19653.788,E2 -19653.788} C_VEL
LIN {X 0,Y 234.514,Z 342.248,A -85,B 0,C 180,E1 -19656.299,E2 -19656.299} C_VEL
LIN {X 0,Y 235.48,Z 334.006,A -85,B 0,C 180,E1 -19658.81,E2 -19658.81} C_VEL
LIN {X 0,Y 236.65,Z 324.885,A -85,B 0,C 180,E1 -19661.065,E2 -19661.065} C_VEL
LIN {X 0,Y 237.855,Z 314.697,A -85,B 0,C 180,E1 -19663.1,E2 -19663.1} C_VEL
LIN {X 0,Y 239.152,Z 303.808,A -85,B 0,C 180,E1 -19664.852,E2 -19664.852} C_VEL
LIN {X 0,Y 240.372,Z 291.535,A -85,B 0,C 180,E1 -19666.424,E2 -19666.424} C_VEL
LIN {X 0,Y 241.603,Z 277.853,A -85,B 0,C 180,E1 -19667.735,E2 -19667.735} C_VEL
LIN {X 0,Y 242.344,Z 264.664,A -85,B 0,C 180,E1 -19668.649,E2 -19668.649} C_VEL
LIN {X 0,Y 243.23,Z 245.008,A -85,B 0,C 180,E1 -19669.488,E2 -19669.488} C_VEL
LIN {X 0,Y 245.719,Z 189.68,A -85,B 0,C 180,E1 -19671.596,E2 -19671.596} C_VEL
LIN {X 0,Y 236.996,Z 165.057,A -85,B 0,C 180,E1 -19673.266,E2 -19673.266} C_VEL
LIN {X 0,Y 234.993,Z 159.215,A -85,B 0,C 180,E1 -19673.719,E2 -19673.719} C_VEL
LIN {X 0,Y 234.958,Z 159.219,A -85,B 0,C 180,E1 -19677.424,E2 -19677.424} C_VEL
LIN {X 0,Y 234.952,Z 159.223,A -85,B 0,C 180,E1 -19681.405,E2 -19681.405} C_VEL
LIN {X 0,Y 234.987,Z 159.217,A -85,B 0,C 180,E1 -19685.246,E2 -19685.246} C_VEL
LIN {X 0,Y 235.005,Z 159.212,A -85,B 0,C 180,E1 -19688.969,E2 -19688.969} C_VEL
LIN {X 0,Y 235.078,Z 159.2,A -85,B 0,C 180,E1 -19694.391,E2 -19694.391} C_VEL
LIN {X 0,Y 235.236,Z 159.181,A -85,B 0,C 180,E1 -19699.673,E2 -19699.673} C_VEL
LIN {X 0,Y 235.401,Z 159.161,A -85,B 0,C 180,E1 -19703.141,E2 -19703.141} C_VEL
LIN {X 0,Y 235.595,Z 159.137,A -85,B 0,C 180,E1 -19708.29,E2 -19708.29} C_VEL
LIN {X 0,Y 235.595,Z 159.135,A -85,B 0,C 180,E1 -19711.709,E2 -19711.709} C_VEL
LIN {X 0,Y 235.401,Z 159.163,A -85,B 0,C 180,E1 -19716.858,E2 -19716.858} C_VEL
LIN {X 0,Y 235.236,Z 159.182,A -85,B 0,C 180,E1 -19720.326,E2 -19720.326} C_VEL
LIN {X 0,Y 235.112,Z 159.197,A -85,B 0,C 180,E1 -19725.606,E2 -19725.606} C_VEL
LIN {X 0,Y 235.006,Z 159.207,A -85,B 0,C 180,E1 -19729.205,E2 -19729.205} C_VEL
LIN {X 0,Y 234.95,Z 159.217,A -85,B 0,C 180,E1 -19732.883,E2 -19732.883} C_VEL
LIN {X 0,Y 234.967,Z 159.214,A -85,B 0,C 180,E1 -19736.657,E2 -19736.657} C_VEL
LIN {X 0,Y 234.93,Z 159.22,A -85,B 0,C 180,E1 -19740.567,E2 -19740.567} C_VEL
LIN {X 0,Y 234.958,Z 159.215,A -85,B 0,C 180,E1 -19744.633,E2 -19744.633} C_VEL
LIN {X 0,Y 234.964,Z 159.215,A -85,B 0,C 180,E1 -19748.952,E2 -19748.952} C_VEL
LIN {X 0,Y 234.963,Z 159.215,A -85,B 0,C 180,E1 -19753.468,E2 -19753.468} C_VEL
LIN {X 0,Y 234.957,Z 159.215,A -85,B 0,C 180,E1 -19756.531,E2 -19756.531} C_VEL
LIN {X 0,Y 234.952,Z 159.216,A -85,B 0,C 180,E1 -19761.086,E2 -19761.086} C_VEL
LIN {X 0,Y 234.957,Z 159.217,A -85,B 0,C 180,E1 -19765.367,E2 -19765.367} C_VEL
LIN {X 0,Y 234.966,Z 159.213,A -85,B 0,C 180,E1 -19770.157,E2 -19770.157} C_VEL
LIN {X 0,Y 234.991,Z 159.213,A -85,B 0,C 180,E1 -19773.794,E2 -19773.794} C_VEL
LIN {X 0,Y 235.009,Z 159.209,A -85,B 0,C 180,E1 -19778.97,E2 -19778.97} C_VEL
LIN {X 0,Y 235.094,Z 159.201,A -85,B 0,C 180,E1 -19783.06,E2 -19783.06} C_VEL
LIN {X 0,Y 235.145,Z 159.19,A -85,B 0,C 180,E1 -19787.924,E2 -19787.924} C_VEL
LIN {X 0,Y 235.374,Z 159.166,A -85,B 0,C 180,E1 -19791.415,E2 -19791.415} C_VEL
LIN {X 0,Y 235.4,Z 159.163,A -85,B 0,C 180,E1 -19793.142,E2 -19793.142} C_VEL
LIN {X 0,Y 235.594,Z 159.136,A -85,B 0,C 180,E1 -19798.291,E2 -19798.291} C_VEL
LIN {X 0,Y 235.595,Z 159.136,A -85,B 0,C 180,E1 -19801.71,E2 -19801.71} C_VEL
LIN {X 0,Y 235.404,Z 159.163,A -85,B 0,C 180,E1 -19806.859,E2 -19806.859} C_VEL
LIN {X 0,Y 235.252,Z 159.181,A -85,B 0,C 180,E1 -19810.326,E2 -19810.326} C_VEL
LIN {X 0,Y 235.113,Z 159.196,A -85,B 0,C 180,E1 -19815.607,E2 -19815.607} C_VEL
LIN {X 0,Y 235.007,Z 159.208,A -85,B 0,C 180,E1 -19819.206,E2 -19819.206} C_VEL
LIN {X 0,Y 234.945,Z 159.217,A -85,B 0,C 180,E1 -19823.027,E2 -19823.027} C_VEL
LIN {X 0,Y 234.969,Z 159.215,A -85,B 0,C 180,E1 -19826.658,E2 -19826.658} C_VEL
LIN {X 0,Y 234.935,Z 159.219,A -85,B 0,C 180,E1 -19830.458,E2 -19830.458} C_VEL
LIN {X 0,Y 234.255,Z 159.311,A -85,B 0,C 180,E1 -19831.887,E2 -19831.887} C_VEL
LIN {X 0,Y 231.443,Z 159.668,A -85,B 0,C 180,E1 -19834.222,E2 -19834.222} C_VEL
LIN {X 0,Y 228.222,Z 160.062,A -85,B 0,C 180,E1 -19837.102,E2 -19837.102} C_VEL
LIN {X 0,Y 227.87,Z 160.099,A -85,B 0,C 180,E1 -19838.099,E2 -19838.099} C_VEL
LIN {X 0,Y 227.864,Z 160.099,A -85,B 0,C 180,E1 -19842.731,E2 -19842.731} C_VEL
LIN {X 0,Y 227.812,Z 160.107,A -85,B 0,C 180,E1 -19847.259,E2 -19847.259} C_VEL
LIN {X 0,Y 227.851,Z 160.106,A -85,B 0,C 180,E1 -19851.911,E2 -19851.911} C_VEL
LIN {X 0,Y 227.974,Z 160.111,A -85,B 0,C 180,E1 -19854.042,E2 -19854.042} C_VEL
LIN {X 0,Y 230.186,Z 171.215,A -85,B 0,C 180,E1 -19858.221,E2 -19858.221} C_VEL
LIN {X 0,Y 231.68,Z 178.362,A -85,B 0,C 180,E1 -19860.756,E2 -19860.756} C_VEL
LIN {X 0,Y 233.111,Z 183.5,A -85,B 0,C 180,E1 -19861.094,E2 -19861.094} C_VEL
LIN {X 0,Y 237.64,Z 232.489,A -85,B 0,C 180,E1 -19863.526,E2 -19863.526} C_VEL
LIN {X 0,Y 235.341,Z 288.35,A -85,B 0,C 180,E1 -19865.816,E2 -19865.816} C_VEL
LIN {X 0,Y 234.318,Z 301.802,A -85,B 0,C 180,E1 -19866.701,E2 -19866.701} C_VEL
LIN {X 0,Y 233.032,Z 314.191,A -85,B 0,C 180,E1 -19867.854,E2 -19867.854} C_VEL
LIN {X 0,Y 231.645,Z 326.303,A -85,B 0,C 180,E1 -19869.348,E2 -19869.348} C_VEL
LIN {X 0,Y 230.149,Z 338.017,A -85,B 0,C 180,E1 -19871.2,E2 -19871.2} C_VEL
LIN {X 0,Y 228.612,Z 349.323,A -85,B 0,C 180,E1 -19873.48,E2 -19873.48} C_VEL
LIN {X 0,Y 227.629,Z 358.16,A -85,B 0,C 180,E1 -19875.701,E2 -19875.701} C_VEL
LIN {X 0,Y 226.749,Z 366.676,A -85,B 0,C 180,E1 -19878.378,E2 -19878.378} C_VEL
LIN {X 0,Y 226.262,Z 373.486,A -85,B 0,C 180,E1 -19881.066,E2 -19881.066} C_VEL
LIN {X 0,Y 226.113,Z 379.373,A -85,B 0,C 180,E1 -19884.058,E2 -19884.058} C_VEL
LIN {X 0,Y 226.069,Z 382.929,A -85,B 0,C 180,E1 -19886.436,E2 -19886.436} C_VEL
LIN {X 0,Y 226.03,Z 384.97,A -85,B 0,C 180,E1 -19888.219,E2 -19888.219} C_VEL
LIN {X 0,Y 226.203,Z 386.565,A -85,B 0,C 180,E1 -19890.001,E2 -19890.001} C_VEL
LIN {X 0,Y 225.898,Z 387.673,A -85,B 0,C 180,E1 -19891.783,E2 -19891.783} C_VEL
LIN {X 0,Y 225.862,Z 388.369,A -85,B 0,C 180,E1 -19893.569,E2 -19893.569} C_VEL
LIN {X 0,Y 225.784,Z 388.447,A -85,B 0,C 180,E1 -19897.153,E2 -19897.153} C_VEL
LIN {X 0,Y 226.483,Z 386.977,A -85,B 0,C 180,E1 -19900.731,E2 -19900.731} C_VEL
LIN {X 0,Y 227.059,Z 385.616,A -85,B 0,C 180,E1 -19902.514,E2 -19902.514} C_VEL
LIN {X 0,Y 228.487,Z 382.83,A -85,B 0,C 180,E1 -19905.157,E2 -19905.157} C_VEL
LIN {X 0,Y 231.256,Z 377.549,A -85,B 0,C 180,E1 -19908.609,E2 -19908.609} C_VEL
LIN {X 0,Y 233.882,Z 371.997,A -85,B 0,C 180,E1 -19911.324,E2 -19911.324} C_VEL
LIN {X 0,Y 237.468,Z 364.766,A -85,B 0,C 180,E1 -19914.013,E2 -19914.013} C_VEL
LIN {X 0,Y 241.185,Z 356.601,A -85,B 0,C 180,E1 -19916.384,E2 -19916.384} C_VEL
LIN {X 0,Y 245.539,Z 346.688,A -85,B 0,C 180,E1 -19918.649,E2 -19918.649} C_VEL
LIN {X 0,Y 249.513,Z 336.506,A -85,B 0,C 180,E1 -19920.465,E2 -19920.465} C_VEL
LIN {X 0,Y 253.284,Z 325.341,A -85,B 0,C 180,E1 -19922.051,E2 -19922.051} C_VEL
LIN {X 0,Y 257.076,Z 312.854,A -85,B 0,C 180,E1 -19923.38,E2 -19923.38} C_VEL
LIN {X 0,Y 260.512,Z 298.757,A -85,B 0,C 180,E1 -19924.509,E2 -19924.509} C_VEL
LIN {X 0,Y 263.049,Z 284.79,A -85,B 0,C 180,E1 -19925.294,E2 -19925.294} C_VEL
LIN {X 0,Y 265.824,Z 259.733,A -85,B 0,C 180,E1 -19926.271,E2 -19926.271} C_VEL
LIN {X 0,Y 267.819,Z 239.86,A -85,B 0,C 180,E1 -19927.04,E2 -19927.04} C_VEL
LIN {X 0,Y 267.074,Z 226.279,A -85,B 0,C 180,E1 -19928.238,E2 -19928.238} C_VEL
LIN {X 0,Y 263.763,Z 217.663,A -85,B 0,C 180,E1 -19930.068,E2 -19930.068} C_VEL
LIN {X 0,Y 260.716,Z 210.844,A -85,B 0,C 180,E1 -19931.893,E2 -19931.893} C_VEL
LIN {X 0,Y 258.368,Z 206.1,A -85,B 0,C 180,E1 -19933.408,E2 -19933.408} C_VEL
LIN {X 0,Y 255.687,Z 200.775,A -85,B 0,C 180,E1 -19935.447,E2 -19935.447} C_VEL
LIN {X 0,Y 252.452,Z 194.852,A -85,B 0,C 180,E1 -19938.427,E2 -19938.427} C_VEL
LIN {X 0,Y 249.128,Z 188.977,A -85,B 0,C 180,E1 -19943.23,E2 -19943.23} C_VEL
LIN {X 0,Y 248.372,Z 187.248,A -85,B 0,C 180,E1 -19945.533,E2 -19945.533} C_VEL
LIN {X 0,Y 248.101,Z 186.507,A -85,B 0,C 180,E1 -19948.193,E2 -19948.193} C_VEL
LIN {X 0,Y 248.702,Z 186.837,A -85,B 0,C 180,E1 -19951.288,E2 -19951.288} C_VEL
LIN {X 0,Y 251.58,Z 189.426,A -85,B 0,C 180,E1 -19955.953,E2 -19955.953} C_VEL
LIN {X 0,Y 255.144,Z 194.018,A -85,B 0,C 180,E1 -19959.479,E2 -19959.479} C_VEL
LIN {X 0,Y 258.265,Z 198.283,A -85,B 0,C 180,E1 -19961.785,E2 -19961.785} C_VEL
LIN {X 0,Y 261.712,Z 203.487,A -85,B 0,C 180,E1 -19963.942,E2 -19963.942} C_VEL
LIN {X 0,Y 265.842,Z 210.425,A -85,B 0,C 180,E1 -19966.194,E2 -19966.194} C_VEL
LIN {X 0,Y 268.39,Z 215.611,A -85,B 0,C 180,E1 -19967.485,E2 -19967.485} C_VEL
LIN {X 0,Y 269.632,Z 218.763,A -85,B 0,C 180,E1 -19968.135,E2 -19968.135} C_VEL
LIN {X 0,Y 264.469,Z 267.025,A -85,B 0,C 180,E1 -19969.973,E2 -19969.973} C_VEL
LIN {X 0,Y 262.538,Z 279.96,A -85,B 0,C 180,E1 -19970.757,E2 -19970.757} C_VEL
LIN {X 0,Y 260.276,Z 291.063,A -85,B 0,C 180,E1 -19971.654,E2 -19971.654} C_VEL
LIN {X 0,Y 257.271,Z 303.052,A -85,B 0,C 180,E1 -19972.938,E2 -19972.938} C_VEL
LIN {X 0,Y 253.773,Z 314.351,A -85,B 0,C 180,E1 -19974.458,E2 -19974.458} C_VEL
LIN {X 0,Y 250.244,Z 324.339,A -85,B 0,C 180,E1 -19976.175,E2 -19976.175} C_VEL
LIN {X 0,Y 246.702,Z 333.115,A -85,B 0,C 180,E1 -19978.078,E2 -19978.078} C_VEL
LIN {X 0,Y 242.732,Z 341.693,A -85,B 0,C 180,E1 -19980.414,E2 -19980.414} C_VEL
LIN {X 0,Y 239.241,Z 348.62,A -85,B 0,C 180,E1 -19982.806,E2 -19982.806} C_VEL
LIN {X 0,Y 236.328,Z 353.857,A -85,B 0,C 180,E1 -19985.118,E2 -19985.118} C_VEL
LIN {X 0,Y 233.863,Z 357.859,A -85,B 0,C 180,E1 -19987.379,E2 -19987.379} C_VEL
LIN {X 0,Y 231.092,Z 361.914,A -85,B 0,C 180,E1 -19990.513,E2 -19990.513} C_VEL
LIN {X 0,Y 229.812,Z 363.557,A -85,B 0,C 180,E1 -19992.36,E2 -19992.36} C_VEL
LIN {X 0,Y 228.655,Z 364.766,A -85,B 0,C 180,E1 -19994.234,E2 -19994.234} C_VEL
LIN {X 0,Y 227.452,Z 365.604,A -85,B 0,C 180,E1 -19996.69,E2 -19996.69} C_VEL
LIN {X 0,Y 226.368,Z 365.52,A -85,B 0,C 180,E1 -19999.968,E2 -19999.968} C_VEL
LIN {X 0,Y 225.949,Z 364.808,A -85,B 0,C 180,E1 -20001.916,E2 -20001.916} C_VEL
LIN {X 0,Y 225.63,Z 362.295,A -85,B 0,C 180,E1 -20005.403,E2 -20005.403} C_VEL
LIN {X 0,Y 225.818,Z 358.515,A -85,B 0,C 180,E1 -20008.621,E2 -20008.621} C_VEL
LIN {X 0,Y 226.298,Z 353.054,A -85,B 0,C 180,E1 -20011.867,E2 -20011.867} C_VEL
LIN {X 0,Y 226.966,Z 346.19,A -85,B 0,C 180,E1 -20014.949,E2 -20014.949} C_VEL
LIN {X 0,Y 227.873,Z 338.473,A -85,B 0,C 180,E1 -20017.646,E2 -20017.646} C_VEL
LIN {X 0,Y 228.987,Z 329.664,A -85,B 0,C 180,E1 -20020.129,E2 -20020.129} C_VEL
LIN {X 0,Y 230.135,Z 320.618,A -85,B 0,C 180,E1 -20022.209,E2 -20022.209} C_VEL
LIN {X 0,Y 231.513,Z 309.411,A -85,B 0,C 180,E1 -20024.282,E2 -20024.282} C_VEL
LIN {X 0,Y 232.884,Z 297.463,A -85,B 0,C 180,E1 -20026.044,E2 -20026.044} C_VEL
LIN {X 0,Y 234.127,Z 284.506,A -85,B 0,C 180,E1 -20027.502,E2 -20027.502} C_VEL
LIN {X 0,Y 235.002,Z 272.258,A -85,B 0,C 180,E1 -20028.544,E2 -20028.544} C_VEL
LIN {X 0,Y 235.802,Z 258.635,A -85,B 0,C 180,E1 -20029.34,E2 -20029.34} C_VEL
LIN {X 0,Y 238.812,Z 190.756,A -85,B 0,C 180,E1 -20032.029,E2 -20032.029} C_VEL
LIN {X 0,Y 228.548,Z 162.194,A -85,B 0,C 180,E1 -20034.057,E2 -20034.057} C_VEL
LIN {X 0,Y 227.935,Z 160.092,A -85,B 0,C 180,E1 -20034.24,E2 -20034.24} C_VEL
LIN {X 0,Y 227.872,Z 160.1,A -85,B 0,C 180,E1 -20038.377,E2 -20038.377} C_VEL
LIN {X 0,Y 227.886,Z 160.099,A -85,B 0,C 180,E1 -20042.444,E2 -20042.444} C_VEL
LIN {X 0,Y 227.913,Z 160.095,A -85,B 0,C 180,E1 -20046.367,E2 -20046.367} C_VEL
LIN {X 0,Y 227.931,Z 160.09,A -85,B 0,C 180,E1 -20050.173,E2 -20050.173} C_VEL
LIN {X 0,Y 228.022,Z 160.079,A -85,B 0,C 180,E1 -20053.895,E2 -20053.895} C_VEL
LIN {X 0,Y 228.067,Z 160.074,A -85,B 0,C 180,E1 -20057.542,E2 -20057.542} C_VEL
LIN {X 0,Y 228.304,Z 160.047,A -85,B 0,C 180,E1 -20061.145,E2 -20061.145} C_VEL
LIN {X 0,Y 228.353,Z 160.041,A -85,B 0,C 180,E1 -20062.928,E2 -20062.928} C_VEL
LIN {X 0,Y 228.554,Z 160.014,A -85,B 0,C 180,E1 -20068.237,E2 -20068.237} C_VEL
LIN {X 0,Y 228.553,Z 160.012,A -85,B 0,C 180,E1 -20071.761,E2 -20071.761} C_VEL
LIN {X 0,Y 228.352,Z 160.04,A -85,B 0,C 180,E1 -20077.071,E2 -20077.071} C_VEL
LIN {X 0,Y 228.161,Z 160.063,A -85,B 0,C 180,E1 -20080.65,E2 -20080.65} C_VEL
LIN {X 0,Y 228.063,Z 160.076,A -85,B 0,C 180,E1 -20084.271,E2 -20084.271} C_VEL
LIN {X 0,Y 228.001,Z 160.083,A -85,B 0,C 180,E1 -20087.953,E2 -20087.953} C_VEL
LIN {X 0,Y 227.914,Z 160.096,A -85,B 0,C 180,E1 -20092.321,E2 -20092.321} C_VEL
LIN {X 0,Y 227.94,Z 160.089,A -85,B 0,C 180,E1 -20096.603,E2 -20096.603} C_VEL
LIN {X 0,Y 227.907,Z 160.097,A -85,B 0,C 180,E1 -20100.296,E2 -20100.296} C_VEL
LIN {X 0,Y 227.887,Z 160.098,A -85,B 0,C 180,E1 -20103.718,E2 -20103.718} C_VEL
LIN {X 0,Y 227.868,Z 160.102,A -85,B 0,C 180,E1 -20108.085,E2 -20108.085} C_VEL
LIN {X 0,Y 227.906,Z 160.093,A -85,B 0,C 180,E1 -20112.719,E2 -20112.719} C_VEL
LIN {X 0,Y 227.895,Z 160.099,A -85,B 0,C 180,E1 -20117.741,E2 -20117.741} C_VEL
LIN {X 0,Y 227.868,Z 160.098,A -85,B 0,C 180,E1 -20121.915,E2 -20121.915} C_VEL
LIN {X 0,Y 227.887,Z 160.097,A -85,B 0,C 180,E1 -20126.373,E2 -20126.373} C_VEL
LIN {X 0,Y 227.916,Z 160.09,A -85,B 0,C 180,E1 -20130.438,E2 -20130.438} C_VEL
LIN {X 0,Y 227.926,Z 160.092,A -85,B 0,C 180,E1 -20134.426,E2 -20134.426} C_VEL
LIN {X 0,Y 227.959,Z 160.085,A -85,B 0,C 180,E1 -20138.288,E2 -20138.288} C_VEL
LIN {X 0,Y 228.032,Z 160.08,A -85,B 0,C 180,E1 -20142.826,E2 -20142.826} C_VEL
LIN {X 0,Y 228.092,Z 160.07,A -85,B 0,C 180,E1 -20147.545,E2 -20147.545} C_VEL
LIN {X 0,Y 228.303,Z 160.048,A -85,B 0,C 180,E1 -20151.147,E2 -20151.147} C_VEL
LIN {X 0,Y 228.352,Z 160.042,A -85,B 0,C 180,E1 -20152.929,E2 -20152.929} C_VEL
LIN {X 0,Y 228.553,Z 160.013,A -85,B 0,C 180,E1 -20158.239,E2 -20158.239} C_VEL
LIN {X 0,Y 228.553,Z 160.013,A -85,B 0,C 180,E1 -20161.763,E2 -20161.763} C_VEL
LIN {X 0,Y 228.357,Z 160.04,A -85,B 0,C 180,E1 -20167.072,E2 -20167.072} C_VEL
LIN {X 0,Y 228.17,Z 160.063,A -85,B 0,C 180,E1 -20170.651,E2 -20170.651} C_VEL
LIN {X 0,Y 228.057,Z 160.077,A -85,B 0,C 180,E1 -20176.103,E2 -20176.103} C_VEL
LIN {X 0,Y 227.937,Z 160.089,A -85,B 0,C 180,E1 -20179.827,E2 -20179.827} C_VEL
LIN {X 0,Y 227.906,Z 160.094,A -85,B 0,C 180,E1 -20183.634,E2 -20183.634} C_VEL
LIN {X 0,Y 227.885,Z 160.096,A -85,B 0,C 180,E1 -20187.556,E2 -20187.556} C_VEL
LIN {X 0,Y 227.873,Z 160.098,A -85,B 0,C 180,E1 -20191.623,E2 -20191.623} C_VEL
LIN {X 0,Y 227.901,Z 160.096,A -85,B 0,C 180,E1 -20195.869,E2 -20195.869} C_VEL
LIN {X 0,Y 227.87,Z 160.099,A -85,B 0,C 180,E1 -20198.099,E2 -20198.099} C_VEL
LIN {X 0,Y 227.152,Z 160.19,A -85,B 0,C 180,E1 -20199.575,E2 -20199.575} C_VEL
LIN {X 0,Y 224.296,Z 160.547,A -85,B 0,C 180,E1 -20201.984,E2 -20201.984} C_VEL
LIN {X 0,Y 221.891,Z 160.845,A -85,B 0,C 180,E1 -20203.949,E2 -20203.949} C_VEL
LIN {X 0,Y 220.849,Z 160.972,A -85,B 0,C 180,E1 -20205.474,E2 -20205.474} C_VEL
LIN {X 0,Y 220.757,Z 160.982,A -85,B 0,C 180,E1 -20205.99,E2 -20205.99} C_VEL
LIN {X 0,Y 220.807,Z 160.979,A -85,B 0,C 180,E1 -20210.464,E2 -20210.464} C_VEL
LIN {X 0,Y 220.897,Z 161.052,A -85,B 0,C 180,E1 -20213.732,E2 -20213.732} C_VEL
LIN {X 0,Y 223.227,Z 172.619,A -85,B 0,C 180,E1 -20218.219,E2 -20218.219} C_VEL
LIN {X 0,Y 224.312,Z 177.788,A -85,B 0,C 180,E1 -20220.15,E2 -20220.15} C_VEL
LIN {X 0,Y 226.375,Z 184.88,A -85,B 0,C 180,E1 -20220.635,E2 -20220.635} C_VEL
LIN {X 0,Y 230.782,Z 232.392,A -85,B 0,C 180,E1 -20223.077,E2 -20223.077} C_VEL
LIN {X 0,Y 228.449,Z 287.42,A -85,B 0,C 180,E1 -20225.401,E2 -20225.401} C_VEL
LIN {X 0,Y 227.424,Z 300.961,A -85,B 0,C 180,E1 -20226.314,E2 -20226.314} C_VEL
LIN {X 0,Y 226.202,Z 312.441,A -85,B 0,C 180,E1 -20227.389,E2 -20227.389} C_VEL
LIN {X 0,Y 224.789,Z 324.799,A -85,B 0,C 180,E1 -20228.928,E2 -20228.928} C_VEL
LIN {X 0,Y 223.23,Z 336.659,A -85,B 0,C 180,E1 -20230.823,E2 -20230.823} C_VEL
LIN {X 0,Y 221.76,Z 347.161,A -85,B 0,C 180,E1 -20232.954,E2 -20232.954} C_VEL
LIN {X 0,Y 220.728,Z 356.278,A -85,B 0,C 180,E1 -20235.244,E2 -20235.244} C_VEL
LIN {X 0,Y 219.894,Z 363.773,A -85,B 0,C 180,E1 -20237.542,E2 -20237.542} C_VEL
LIN {X 0,Y 219.303,Z 371.109,A -85,B 0,C 180,E1 -20240.315,E2 -20240.315} C_VEL
LIN {X 0,Y 219.074,Z 376.024,A -85,B 0,C 180,E1 -20242.628,E2 -20242.628} C_VEL
LIN {X 0,Y 219.08,Z 380.711,A -85,B 0,C 180,E1 -20245.401,E2 -20245.401} C_VEL
LIN {X 0,Y 218.964,Z 384.146,A -85,B 0,C 180,E1 -20248.161,E2 -20248.161} C_VEL
LIN {X 0,Y 219.145,Z 385.828,A -85,B 0,C 180,E1 -20250.001,E2 -20250.001} C_VEL
LIN {X 0,Y 218.829,Z 387.01,A -85,B 0,C 180,E1 -20251.841,E2 -20251.841} C_VEL
LIN {X 0,Y 218.786,Z 387.79,A -85,B 0,C 180,E1 -20253.684,E2 -20253.684} C_VEL
LIN {X 0,Y 218.625,Z 388.143,A -85,B 0,C 180,E1 -20255.535,E2 -20255.535} C_VEL
LIN {X 0,Y 218.995,Z 387.611,A -85,B 0,C 180,E1 -20259.234,E2 -20259.234} C_VEL
LIN {X 0,Y 220.09,Z 385.526,A -85,B 0,C 180,E1 -20262.917,E2 -20262.917} C_VEL
LIN {X 0,Y 221.635,Z 382.893,A -85,B 0,C 180,E1 -20265.637,E2 -20265.637} C_VEL
LIN {X 0,Y 223.737,Z 379.309,A -85,B 0,C 180,E1 -20268.308,E2 -20268.308} C_VEL
LIN {X 0,Y 226.301,Z 374.386,A -85,B 0,C 180,E1 -20271.101,E2 -20271.101} C_VEL
LIN {X 0,Y 229.858,Z 367.878,A -85,B 0,C 180,E1 -20273.9,E2 -20273.9} C_VEL
LIN {X 0,Y 233.646,Z 360.585,A -85,B 0,C 180,E1 -20276.339,E2 -20276.339} C_VEL
LIN {X 0,Y 237.105,Z 353.306,A -85,B 0,C 180,E1 -20278.311,E2 -20278.311} C_VEL
LIN {X 0,Y 241.04,Z 344.584,A -85,B 0,C 180,E1 -20280.196,E2 -20280.196} C_VEL
LIN {X 0,Y 245.692,Z 332.972,A -85,B 0,C 180,E1 -20282.193,E2 -20282.193} C_VEL
LIN {X 0,Y 249.372,Z 322.617,A -85,B 0,C 180,E1 -20283.58,E2 -20283.58} C_VEL
LIN {X 0,Y 253.388,Z 309.587,A -85,B 0,C 180,E1 -20284.894,E2 -20284.894} C_VEL
LIN {X 0,Y 256.211,Z 298.2,A -85,B 0,C 180,E1 -20285.776,E2 -20285.776} C_VEL
LIN {X 0,Y 258.807,Z 284.264,A -85,B 0,C 180,E1 -20286.565,E2 -20286.565} C_VEL
LIN {X 0,Y 262.233,Z 254.774,A -85,B 0,C 180,E1 -20287.716,E2 -20287.716} C_VEL
LIN {X 0,Y 263.67,Z 241.209,A -85,B 0,C 180,E1 -20288.26,E2 -20288.26} C_VEL
LIN {X 0,Y 263.235,Z 230.2,A -85,B 0,C 180,E1 -20289.261,E2 -20289.261} C_VEL
LIN {X 0,Y 260.526,Z 222.721,A -85,B 0,C 180,E1 -20290.896,E2 -20290.896} C_VEL
LIN {X 0,Y 257.866,Z 216.478,A -85,B 0,C 180,E1 -20292.618,E2 -20292.618} C_VEL
LIN {X 0,Y 255.779,Z 211.926,A -85,B 0,C 180,E1 -20294.113,E2 -20294.113} C_VEL
LIN {X 0,Y 253.413,Z 207.034,A -85,B 0,C 180,E1 -20296.01,E2 -20296.01} C_VEL
LIN {X 0,Y 250.481,Z 201.37,A -85,B 0,C 180,E1 -20298.934,E2 -20298.934} C_VEL
LIN {X 0,Y 247.596,Z 195.716,A -85,B 0,C 180,E1 -20303.613,E2 -20303.613} C_VEL
LIN {X 0,Y 246.953,Z 194.046,A -85,B 0,C 180,E1 -20305.965,E2 -20305.965} C_VEL
LIN {X 0,Y 246.881,Z 193.44,A -85,B 0,C 180,E1 -20309.175,E2 -20309.175} C_VEL
LIN {X 0,Y 247.672,Z 194.132,A -85,B 0,C 180,E1 -20312.064,E2 -20312.064} C_VEL
LIN {X 0,Y 250.097,Z 196.539,A -85,B 0,C 180,E1 -20315.897,E2 -20315.897} C_VEL
LIN {X 0,Y 253.178,Z 200.568,A -85,B 0,C 180,E1 -20319.051,E2 -20319.051} C_VEL
LIN {X 0,Y 255.998,Z 204.585,A -85,B 0,C 180,E1 -20321.269,E2 -20321.269} C_VEL
LIN {X 0,Y 259.071,Z 209.507,A -85,B 0,C 180,E1 -20323.347,E2 -20323.347} C_VEL
LIN {X 0,Y 263.242,Z 216.819,A -85,B 0,C 180,E1 -20325.761,E2 -20325.761} C_VEL
LIN {X 0,Y 265.461,Z 221.798,A -85,B 0,C 180,E1 -20326.954,E2 -20326.954} C_VEL
LIN {X 0,Y 260.203,Z 267.652,A -85,B 0,C 180,E1 -20328.741,E2 -20328.741} C_VEL
LIN {X 0,Y 258.226,Z 280.249,A -85,B 0,C 180,E1 -20329.509,E2 -20329.509} C_VEL
LIN {X 0,Y 255.623,Z 292.453,A -85,B 0,C 180,E1 -20330.504,E2 -20330.504} C_VEL
LIN {X 0,Y 252.459,Z 304.26,A -85,B 0,C 180,E1 -20331.797,E2 -20331.797} C_VEL
LIN {X 0,Y 248.846,Z 315.207,A -85,B 0,C 180,E1 -20333.309,E2 -20333.309} C_VEL
LIN {X 0,Y 245.048,Z 325.168,A -85,B 0,C 180,E1 -20335.064,E2 -20335.064} C_VEL
LIN {X 0,Y 241.192,Z 334.127,A -85,B 0,C 180,E1 -20337.048,E2 -20337.048} C_VEL
LIN {X 0,Y 237.497,Z 341.748,A -85,B 0,C 180,E1 -20339.152,E2 -20339.152} C_VEL
LIN {X 0,Y 233.485,Z 349.102,A -85,B 0,C 180,E1 -20341.724,E2 -20341.724} C_VEL
LIN {X 0,Y 229.982,Z 354.891,A -85,B 0,C 180,E1 -20344.381,E2 -20344.381} C_VEL
LIN {X 0,Y 226.737,Z 359.643,A -85,B 0,C 180,E1 -20347.302,E2 -20347.302} C_VEL
LIN {X 0,Y 225.192,Z 361.707,A -85,B 0,C 180,E1 -20348.977,E2 -20348.977} C_VEL
LIN {X 0,Y 222.83,Z 364.462,A -85,B 0,C 180,E1 -20352.111,E2 -20352.111} C_VEL
LIN {X 0,Y 221.253,Z 365.738,A -85,B 0,C 180,E1 -20354.721,E2 -20354.721} C_VEL
LIN {X 0,Y 220.29,Z 366.181,A -85,B 0,C 180,E1 -20356.841,E2 -20356.841} C_VEL
LIN {X 0,Y 219.656,Z 366.092,A -85,B 0,C 180,E1 -20358.659,E2 -20358.659} C_VEL
LIN {X 0,Y 218.934,Z 365.226,A -85,B 0,C 180,E1 -20361.419,E2 -20361.419} C_VEL
LIN {X 0,Y 218.566,Z 362.971,A -85,B 0,C 180,E1 -20364.709,E2 -20364.709} C_VEL
LIN {X 0,Y 218.625,Z 359.64,A -85,B 0,C 180,E1 -20367.782,E2 -20367.782} C_VEL
LIN {X 0,Y 219.014,Z 354.936,A -85,B 0,C 180,E1 -20370.892,E2 -20370.892} C_VEL
LIN {X 0,Y 219.554,Z 349.404,A -85,B 0,C 180,E1 -20373.667,E2 -20373.667} C_VEL
LIN {X 0,Y 220.43,Z 341.742,A -85,B 0,C 180,E1 -20376.679,E2 -20376.679} C_VEL
LIN {X 0,Y 221.475,Z 333.085,A -85,B 0,C 180,E1 -20379.393,E2 -20379.393} C_VEL
LIN {X 0,Y 222.729,Z 323.462,A -85,B 0,C 180,E1 -20381.803,E2 -20381.803} C_VEL
LIN {X 0,Y 223.948,Z 313.699,A -85,B 0,C 180,E1 -20383.796,E2 -20383.796} C_VEL
LIN {X 0,Y 225.33,Z 302.416,A -85,B 0,C 180,E1 -20385.66,E2 -20385.66} C_VEL
LIN {X 0,Y 226.661,Z 289.693,A -85,B 0,C 180,E1 -20387.297,E2 -20387.297} C_VEL
LIN {X 0,Y 227.854,Z 276.478,A -85,B 0,C 180,E1 -20388.581,E2 -20388.581} C_VEL
LIN {X 0,Y 228.658,Z 262.67,A -85,B 0,C 180,E1 -20389.526,E2 -20389.526} C_VEL
LIN {X 0,Y 231.945,Z 192.113,A -85,B 0,C 180,E1 -20392.471,E2 -20392.471} C_VEL
LIN {X 0,Y 222.332,Z 165.351,A -85,B 0,C 180,E1 -20394.42,E2 -20394.42} C_VEL
LIN {X 0,Y 220.895,Z 160.968,A -85,B 0,C 180,E1 -20394.783,E2 -20394.783} C_VEL
LIN {X 0,Y 220.868,Z 160.976,A -85,B 0,C 180,E1 -20399.394,E2 -20399.394} C_VEL
LIN {X 0,Y 220.895,Z 160.972,A -85,B 0,C 180,E1 -20403.549,E2 -20403.549} C_VEL
LIN {X 0,Y 220.877,Z 160.972,A -85,B 0,C 180,E1 -20407.553,E2 -20407.553} C_VEL
LIN {X 0,Y 220.929,Z 160.964,A -85,B 0,C 180,E1 -20412.616,E2 -20412.616} C_VEL
LIN {X 0,Y 221.003,Z 160.955,A -85,B 0,C 180,E1 -20417.137,E2 -20417.137} C_VEL
LIN {X 0,Y 221.235,Z 160.928,A -85,B 0,C 180,E1 -20420.86,E2 -20420.86} C_VEL
LIN {X 0,Y 221.288,Z 160.92,A -85,B 0,C 180,E1 -20422.701,E2 -20422.701} C_VEL
LIN {X 0,Y 221.512,Z 160.891,A -85,B 0,C 180,E1 -20428.181,E2 -20428.181} C_VEL
LIN {X 0,Y 221.511,Z 160.889,A -85,B 0,C 180,E1 -20431.817,E2 -20431.817} C_VEL
LIN {X 0,Y 221.287,Z 160.919,A -85,B 0,C 180,E1 -20437.298,E2 -20437.298} C_VEL
LIN {X 0,Y 221.11,Z 160.939,A -85,B 0,C 180,E1 -20440.994,E2 -20440.994} C_VEL
LIN {X 0,Y 221.014,Z 160.955,A -85,B 0,C 180,E1 -20446.629,E2 -20446.629} C_VEL
LIN {X 0,Y 220.882,Z 160.97,A -85,B 0,C 180,E1 -20450.486,E2 -20450.486} C_VEL
LIN {X 0,Y 220.86,Z 160.974,A -85,B 0,C 180,E1 -20454.435,E2 -20454.435} C_VEL
LIN {X 0,Y 220.835,Z 160.975,A -85,B 0,C 180,E1 -20458.513,E2 -20458.513} C_VEL
LIN {X 0,Y 220.822,Z 160.977,A -85,B 0,C 180,E1 -20462.754,E2 -20462.754} C_VEL
LIN {X 0,Y 220.835,Z 160.973,A -85,B 0,C 180,E1 -20467.288,E2 -20467.288} C_VEL
LIN {X 0,Y 220.85,Z 160.975,A -85,B 0,C 180,E1 -20471.933,E2 -20471.933} C_VEL
LIN {X 0,Y 220.858,Z 160.972,A -85,B 0,C 180,E1 -20477.044,E2 -20477.044} C_VEL
LIN {X 0,Y 220.848,Z 160.973,A -85,B 0,C 180,E1 -20480.473,E2 -20480.473} C_VEL
LIN {X 0,Y 220.813,Z 160.977,A -85,B 0,C 180,E1 -20485.048,E2 -20485.048} C_VEL
LIN {X 0,Y 220.865,Z 160.974,A -85,B 0,C 180,E1 -20489.395,E2 -20489.395} C_VEL
LIN {X 0,Y 220.893,Z 160.971,A -85,B 0,C 180,E1 -20493.55,E2 -20493.55} C_VEL
LIN {X 0,Y 220.875,Z 160.97,A -85,B 0,C 180,E1 -20497.554,E2 -20497.554} C_VEL
LIN {X 0,Y 220.982,Z 160.957,A -85,B 0,C 180,E1 -20502.571,E2 -20502.571} C_VEL
LIN {X 0,Y 221.024,Z 160.952,A -85,B 0,C 180,E1 -20507.14,E2 -20507.14} C_VEL
LIN {X 0,Y 221.234,Z 160.927,A -85,B 0,C 180,E1 -20510.861,E2 -20510.861} C_VEL
LIN {X 0,Y 221.287,Z 160.921,A -85,B 0,C 180,E1 -20512.702,E2 -20512.702} C_VEL
LIN {X 0,Y 221.511,Z 160.89,A -85,B 0,C 180,E1 -20518.183,E2 -20518.183} C_VEL
LIN {X 0,Y 221.511,Z 160.89,A -85,B 0,C 180,E1 -20521.819,E2 -20521.819} C_VEL
LIN {X 0,Y 221.31,Z 160.916,A -85,B 0,C 180,E1 -20527.298,E2 -20527.298} C_VEL
LIN {X 0,Y 221.116,Z 160.939,A -85,B 0,C 180,E1 -20530.995,E2 -20530.995} C_VEL
LIN {X 0,Y 221.016,Z 160.955,A -85,B 0,C 180,E1 -20536.631,E2 -20536.631} C_VEL
LIN {X 0,Y 220.884,Z 160.969,A -85,B 0,C 180,E1 -20540.488,E2 -20540.488} C_VEL
LIN {X 0,Y 220.861,Z 160.975,A -85,B 0,C 180,E1 -20544.436,E2 -20544.436} C_VEL
LIN {X 0,Y 220.836,Z 160.974,A -85,B 0,C 180,E1 -20548.514,E2 -20548.514} C_VEL
LIN {X 0,Y 220.824,Z 160.977,A -85,B 0,C 180,E1 -20552.756,E2 -20552.756} C_VEL
LIN {X 0,Y 220.838,Z 160.971,A -85,B 0,C 180,E1 -20557.289,E2 -20557.289} C_VEL
LIN {X 0,Y 220.815,Z 160.981,A -85,B 0,C 180,E1 -20561.943,E2 -20561.943} C_VEL
LIN {X 0,Y 220.757,Z 160.982,A -85,B 0,C 180,E1 -20565.99,E2 -20565.99} C_VEL
LIN {X 0,Y 220.054,Z 161.073,A -85,B 0,C 180,E1 -20567.004,E2 -20567.004} C_VEL
LIN {X 0,Y 217.185,Z 161.431,A -85,B 0,C 180,E1 -20568.597,E2 -20568.597} C_VEL
LIN {X 0,Y 214.347,Z 161.785,A -85,B 0,C 180,E1 -20570.231,E2 -20570.231} C_VEL
LIN {X 0,Y 213.732,Z 161.861,A -85,B 0,C 180,E1 -20571.29,E2 -20571.29} C_VEL
LIN {X 0,Y 213.848,Z 161.891,A -85,B 0,C 180,E1 -20573.379,E2 -20573.379} C_VEL
LIN {X 0,Y 216.039,Z 172.824,A -85,B 0,C 180,E1 -20577.76,E2 -20577.76} C_VEL
LIN {X 0,Y 217.066,Z 177.579,A -85,B 0,C 180,E1 -20579.546,E2 -20579.546} C_VEL
LIN {X 0,Y 219.718,Z 187.187,A -85,B 0,C 180,E1 -20580.219,E2 -20580.219} C_VEL
LIN {X 0,Y 223.859,Z 233.616,A -85,B 0,C 180,E1 -20582.683,E2 -20582.683} C_VEL
LIN {X 0,Y 221.488,Z 287.732,A -85,B 0,C 180,E1 -20585.076,E2 -20585.076} C_VEL
LIN {X 0,Y 220.424,Z 301.034,A -85,B 0,C 180,E1 -20586.014,E2 -20586.014} C_VEL
LIN {X 0,Y 219.188,Z 312.391,A -85,B 0,C 180,E1 -20587.123,E2 -20587.123} C_VEL
LIN {X 0,Y 217.75,Z 324.663,A -85,B 0,C 180,E1 -20588.71,E2 -20588.71} C_VEL
LIN {X 0,Y 216.152,Z 336.691,A -85,B 0,C 180,E1 -20590.705,E2 -20590.705} C_VEL
LIN {X 0,Y 214.668,Z 346.931,A -85,B 0,C 180,E1 -20592.864,E2 -20592.864} C_VEL
LIN {X 0,Y 213.645,Z 356.03,A -85,B 0,C 180,E1 -20595.231,E2 -20595.231} C_VEL
LIN {X 0,Y 212.808,Z 363.502,A -85,B 0,C 180,E1 -20597.605,E2 -20597.605} C_VEL
LIN {X 0,Y 212.236,Z 370.808,A -85,B 0,C 180,E1 -20600.47,E2 -20600.47} C_VEL
LIN {X 0,Y 211.999,Z 376.557,A -85,B 0,C 180,E1 -20603.339,E2 -20603.339} C_VEL
LIN {X 0,Y 211.968,Z 380.983,A -85,B 0,C 180,E1 -20606.199,E2 -20606.199} C_VEL
LIN {X 0,Y 211.907,Z 383.242,A -85,B 0,C 180,E1 -20608.1,E2 -20608.1} C_VEL
LIN {X 0,Y 212.087,Z 385.059,A -85,B 0,C 180,E1 -20610.001,E2 -20610.001} C_VEL
LIN {X 0,Y 211.711,Z 387.176,A -85,B 0,C 180,E1 -20613.808,E2 -20613.808} C_VEL
LIN {X 0,Y 211.643,Z 387.673,A -85,B 0,C 180,E1 -20617.634,E2 -20617.634} C_VEL
LIN {X 0,Y 211.975,Z 387.316,A -85,B 0,C 180,E1 -20619.543,E2 -20619.543} C_VEL
LIN {X 0,Y 213.135,Z 385.413,A -85,B 0,C 180,E1 -20623.346,E2 -20623.346} C_VEL
LIN {X 0,Y 214.158,Z 383.889,A -85,B 0,C 180,E1 -20625.221,E2 -20625.221} C_VEL
LIN {X 0,Y 216.227,Z 380.801,A -85,B 0,C 180,E1 -20627.986,E2 -20627.986} C_VEL
LIN {X 0,Y 218.627,Z 376.735,A -85,B 0,C 180,E1 -20630.709,E2 -20630.709} C_VEL
LIN {X 0,Y 221.641,Z 371.639,A -85,B 0,C 180,E1 -20633.352,E2 -20633.352} C_VEL
LIN {X 0,Y 226.017,Z 364.152,A -85,B 0,C 180,E1 -20636.303,E2 -20636.303} C_VEL
LIN {X 0,Y 230.221,Z 356.118,A -85,B 0,C 180,E1 -20638.739,E2 -20638.739} C_VEL
LIN {X 0,Y 235.072,Z 346.366,A -85,B 0,C 180,E1 -20641.047,E2 -20641.047} C_VEL
LIN {X 0,Y 239.898,Z 335.339,A -85,B 0,C 180,E1 -20643.069,E2 -20643.069} C_VEL
LIN {X 0,Y 244.141,Z 324.21,A -85,B 0,C 180,E1 -20644.649,E2 -20644.649} C_VEL
LIN {X 0,Y 248.299,Z 311.788,A -85,B 0,C 180,E1 -20645.968,E2 -20645.968} C_VEL
LIN {X 0,Y 251.764,Z 298.969,A -85,B 0,C 180,E1 -20647.008,E2 -20647.008} C_VEL
LIN {X 0,Y 254.554,Z 285.51,A -85,B 0,C 180,E1 -20647.806,E2 -20647.806} C_VEL
LIN {X 0,Y 257.035,Z 266.583,A -85,B 0,C 180,E1 -20648.582,E2 -20648.582} C_VEL
LIN {X 0,Y 259.74,Z 242.757,A -85,B 0,C 180,E1 -20649.517,E2 -20649.517} C_VEL
LIN {X 0,Y 259.435,Z 233.751,A -85,B 0,C 180,E1 -20650.367,E2 -20650.367} C_VEL
LIN {X 0,Y 256.739,Z 226.117,A -85,B 0,C 180,E1 -20652.2,E2 -20652.2} C_VEL
LIN {X 0,Y 254.776,Z 221.378,A -85,B 0,C 180,E1 -20653.601,E2 -20653.601} C_VEL
LIN {X 0,Y 253.167,Z 217.596,A -85,B 0,C 180,E1 -20654.887,E2 -20654.887} C_VEL
LIN {X 0,Y 251.126,Z 213.118,A -85,B 0,C 180,E1 -20656.689,E2 -20656.689} C_VEL
LIN {X 0,Y 248.603,Z 207.853,A -85,B 0,C 180,E1 -20659.442,E2 -20659.442} C_VEL
LIN {X 0,Y 246.064,Z 202.505,A -85,B 0,C 180,E1 -20663.938,E2 -20663.938} C_VEL
LIN {X 0,Y 245.549,Z 200.967,A -85,B 0,C 180,E1 -20666.102,E2 -20666.102} C_VEL
LIN {X 0,Y 245.504,Z 200.396,A -85,B 0,C 180,E1 -20669.184,E2 -20669.184} C_VEL
LIN {X 0,Y 246.205,Z 201.035,A -85,B 0,C 180,E1 -20671.883,E2 -20671.883} C_VEL
LIN {X 0,Y 248.444,Z 203.328,A -85,B 0,C 180,E1 -20675.605,E2 -20675.605} C_VEL
LIN {X 0,Y 251.202,Z 207.079,A -85,B 0,C 180,E1 -20678.595,E2 -20678.595} C_VEL
LIN {X 0,Y 253.843,Z 211.11,A -85,B 0,C 180,E1 -20680.831,E2 -20680.831} C_VEL
LIN {X 0,Y 256.876,Z 216.138,A -85,B 0,C 180,E1 -20682.995,E2 -20682.995} C_VEL
LIN {X 0,Y 260.615,Z 223.232,A -85,B 0,C 180,E1 -20685.28,E2 -20685.28} C_VEL
LIN {X 0,Y 261.408,Z 225.337,A -85,B 0,C 180,E1 -20685.777,E2 -20685.777} C_VEL
LIN {X 0,Y 256.302,Z 267.902,A -85,B 0,C 180,E1 -20687.428,E2 -20687.428} C_VEL
LIN {X 0,Y 254.087,Z 281.018,A -85,B 0,C 180,E1 -20688.229,E2 -20688.229} C_VEL
LIN {X 0,Y 251.182,Z 293.658,A -85,B 0,C 180,E1 -20689.286,E2 -20689.286} C_VEL
LIN {X 0,Y 247.283,Z 306.966,A -85,B 0,C 180,E1 -20690.8,E2 -20690.8} C_VEL
LIN {X 0,Y 243.493,Z 317.55,A -85,B 0,C 180,E1 -20692.328,E2 -20692.328} C_VEL
LIN {X 0,Y 239.538,Z 327.179,A -85,B 0,C 180,E1 -20694.113,E2 -20694.113} C_VEL
LIN {X 0,Y 235.432,Z 335.93,A -85,B 0,C 180,E1 -20696.148,E2 -20696.148} C_VEL
LIN {X 0,Y 231.609,Z 343.191,A -85,B 0,C 180,E1 -20698.26,E2 -20698.26} C_VEL
LIN {X 0,Y 228.045,Z 349.278,A -85,B 0,C 180,E1 -20700.441,E2 -20700.441} C_VEL
LIN {X 0,Y 224.56,Z 354.679,A -85,B 0,C 180,E1 -20702.899,E2 -20702.899} C_VEL
LIN {X 0,Y 221.47,Z 358.992,A -85,B 0,C 180,E1 -20705.462,E2 -20705.462} C_VEL
LIN {X 0,Y 219.465,Z 361.482,A -85,B 0,C 180,E1 -20707.359,E2 -20707.359} C_VEL
LIN {X 0,Y 217.758,Z 363.446,A -85,B 0,C 180,E1 -20709.286,E2 -20709.286} C_VEL
LIN {X 0,Y 215.665,Z 365.46,A -85,B 0,C 180,E1 -20712.139,E2 -20712.139} C_VEL
LIN {X 0,Y 213.858,Z 366.525,A -85,B 0,C 180,E1 -20715.242,E2 -20715.242} C_VEL
LIN {X 0,Y 213.001,Z 366.636,A -85,B 0,C 180,E1 -20717.274,E2 -20717.274} C_VEL
LIN {X 0,Y 212.344,Z 366.248,A -85,B 0,C 180,E1 -20719.327,E2 -20719.327} C_VEL
LIN {X 0,Y 211.781,Z 365.228,A -85,B 0,C 180,E1 -20721.69,E2 -20721.69} C_VEL
LIN {X 0,Y 211.541,Z 364.035,A -85,B 0,C 180,E1 -20723.495,E2 -20723.495} C_VEL
LIN {X 0,Y 211.452,Z 361.517,A -85,B 0,C 180,E1 -20726.181,E2 -20726.181} C_VEL
LIN {X 0,Y 211.661,Z 358.228,A -85,B 0,C 180,E1 -20728.78,E2 -20728.78} C_VEL
LIN {X 0,Y 212.124,Z 352.868,A -85,B 0,C 180,E1 -20732.012,E2 -20732.012} C_VEL
LIN {X 0,Y 212.733,Z 347.042,A -85,B 0,C 180,E1 -20734.74,E2 -20734.74} C_VEL
LIN {X 0,Y 213.716,Z 338.542,A -85,B 0,C 180,E1 -20737.885,E2 -20737.885} C_VEL
LIN {X 0,Y 214.885,Z 329.509,A -85,B 0,C 180,E1 -20740.543,E2 -20740.543} C_VEL
LIN {X 0,Y 216.268,Z 318.884,A -85,B 0,C 180,E1 -20743.033,E2 -20743.033} C_VEL
LIN {X 0,Y 217.66,Z 308.176,A -85,B 0,C 180,E1 -20745.054,E2 -20745.054} C_VEL
LIN {X 0,Y 219.089,Z 295.994,A -85,B 0,C 180,E1 -20746.867,E2 -20746.867} C_VEL
LIN {X 0,Y 220.292,Z 283.688,A -85,B 0,C 180,E1 -20748.293,E2 -20748.293} C_VEL
LIN {X 0,Y 221.201,Z 271.112,A -85,B 0,C 180,E1 -20749.381,E2 -20749.381} C_VEL
LIN {X 0,Y 222.028,Z 257.322,A -85,B 0,C 180,E1 -20750.19,E2 -20750.19} C_VEL
LIN {X 0,Y 225.073,Z 193.316,A -85,B 0,C 180,E1 -20752.911,E2 -20752.911} C_VEL
LIN {X 0,Y 213.838,Z 161.849,A -85,B 0,C 180,E1 -20755.312,E2 -20755.312} C_VEL
LIN {X 0,Y 213.781,Z 161.857,A -85,B 0,C 180,E1 -20760.453,E2 -20760.453} C_VEL
LIN {X 0,Y 213.801,Z 161.853,A -85,B 0,C 180,E1 -20764.701,E2 -20764.701} C_VEL
LIN {X 0,Y 213.808,Z 161.852,A -85,B 0,C 180,E1 -20768.802,E2 -20768.802} C_VEL
LIN {X 0,Y 213.892,Z 161.841,A -85,B 0,C 180,E1 -20772.799,E2 -20772.799} C_VEL
LIN {X 0,Y 213.942,Z 161.832,A -85,B 0,C 180,E1 -20776.705,E2 -20776.705} C_VEL
LIN {X 0,Y 214.166,Z 161.807,A -85,B 0,C 180,E1 -20780.556,E2 -20780.556} C_VEL
LIN {X 0,Y 214.226,Z 161.799,A -85,B 0,C 180,E1 -20782.459,E2 -20782.459} C_VEL
LIN {X 0,Y 214.445,Z 161.771,A -85,B 0,C 180,E1 -20788.121,E2 -20788.121} C_VEL
LIN {X 0,Y 214.549,Z 161.758,A -85,B 0,C 180,E1 -20789.999,E2 -20789.999} C_VEL
LIN {X 0,Y 214.444,Z 161.769,A -85,B 0,C 180,E1 -20791.877,E2 -20791.877} C_VEL
LIN {X 0,Y 214.225,Z 161.798,A -85,B 0,C 180,E1 -20797.54,E2 -20797.54} C_VEL
LIN {X 0,Y 214.043,Z 161.818,A -85,B 0,C 180,E1 -20801.361,E2 -20801.361} C_VEL
LIN {X 0,Y 213.932,Z 161.835,A -85,B 0,C 180,E1 -20805.236,E2 -20805.236} C_VEL
LIN {X 0,Y 213.833,Z 161.844,A -85,B 0,C 180,E1 -20809.187,E2 -20809.187} C_VEL
LIN {X 0,Y 213.808,Z 161.85,A -85,B 0,C 180,E1 -20813.231,E2 -20813.231} C_VEL
LIN {X 0,Y 213.826,Z 161.846,A -85,B 0,C 180,E1 -20817.449,E2 -20817.449} C_VEL
LIN {X 0,Y 213.777,Z 161.856,A -85,B 0,C 180,E1 -20821.735,E2 -20821.735} C_VEL
LIN {X 0,Y 213.752,Z 161.857,A -85,B 0,C 180,E1 -20826.286,E2 -20826.286} C_VEL
LIN {X 0,Y 213.791,Z 161.853,A -85,B 0,C 180,E1 -20831.106,E2 -20831.106} C_VEL
LIN {X 0,Y 213.805,Z 161.852,A -85,B 0,C 180,E1 -20833.685,E2 -20833.685} C_VEL
LIN {X 0,Y 213.808,Z 161.85,A -85,B 0,C 180,E1 -20836.349,E2 -20836.349} C_VEL
LIN {X 0,Y 213.776,Z 161.855,A -85,B 0,C 180,E1 -20841.346,E2 -20841.346} C_VEL
LIN {X 0,Y 213.767,Z 161.857,A -85,B 0,C 180,E1 -20846.021,E2 -20846.021} C_VEL
LIN {X 0,Y 213.778,Z 161.851,A -85,B 0,C 180,E1 -20850.454,E2 -20850.454} C_VEL
LIN {X 0,Y 213.799,Z 161.852,A -85,B 0,C 180,E1 -20854.702,E2 -20854.702} C_VEL
LIN {X 0,Y 213.81,Z 161.849,A -85,B 0,C 180,E1 -20858.804,E2 -20858.804} C_VEL
LIN {X 0,Y 213.941,Z 161.835,A -85,B 0,C 180,E1 -20862.804,E2 -20862.804} C_VEL
LIN {X 0,Y 213.978,Z 161.829,A -85,B 0,C 180,E1 -20866.709,E2 -20866.709} C_VEL
LIN {X 0,Y 214.165,Z 161.806,A -85,B 0,C 180,E1 -20870.557,E2 -20870.557} C_VEL
LIN {X 0,Y 214.225,Z 161.799,A -85,B 0,C 180,E1 -20872.46,E2 -20872.46} C_VEL
LIN {X 0,Y 214.444,Z 161.77,A -85,B 0,C 180,E1 -20878.123,E2 -20878.123} C_VEL
LIN {X 0,Y 214.549,Z 161.758,A -85,B 0,C 180,E1 -20880.001,E2 -20880.001} C_VEL
LIN {X 0,Y 214.445,Z 161.77,A -85,B 0,C 180,E1 -20881.879,E2 -20881.879} C_VEL
LIN {X 0,Y 214.247,Z 161.796,A -85,B 0,C 180,E1 -20887.54,E2 -20887.54} C_VEL
LIN {X 0,Y 214.046,Z 161.818,A -85,B 0,C 180,E1 -20891.363,E2 -20891.363} C_VEL
LIN {X 0,Y 213.933,Z 161.835,A -85,B 0,C 180,E1 -20895.238,E2 -20895.238} C_VEL
LIN {X 0,Y 213.835,Z 161.845,A -85,B 0,C 180,E1 -20899.188,E2 -20899.188} C_VEL
LIN {X 0,Y 213.81,Z 161.85,A -85,B 0,C 180,E1 -20903.232,E2 -20903.232} C_VEL
LIN {X 0,Y 213.828,Z 161.847,A -85,B 0,C 180,E1 -20907.451,E2 -20907.451} C_VEL
LIN {X 0,Y 213.779,Z 161.854,A -85,B 0,C 180,E1 -20911.736,E2 -20911.736} C_VEL
LIN {X 0,Y 213.754,Z 161.856,A -85,B 0,C 180,E1 -20916.287,E2 -20916.287} C_VEL
LIN {X 0,Y 213.74,Z 161.859,A -85,B 0,C 180,E1 -20921.12,E2 -20921.12} C_VEL
LIN {X 0,Y 213.775,Z 161.856,A -85,B 0,C 180,E1 -20923.677,E2 -20923.677} C_VEL
LIN {X 0,Y 213.713,Z 161.863,A -85,B 0,C 180,E1 -20928.876,E2 -20928.876} C_VEL
LIN {X 0,Y 213.732,Z 161.861,A -85,B 0,C 180,E1 -20931.29,E2 -20931.29} C_VEL
LIN {X 0,Y 213.549,Z 162.292,A -85,B 0,C 180,E1 -20932.324,E2 -20932.324} C_VEL
LIN {X 0,Y 212.596,Z 164.187,A -85,B 0,C 180,E1 -20933.799,E2 -20933.799} C_VEL
LIN {X 0,Y 211.069,Z 167.692,A -85,B 0,C 180,E1 -20935.395,E2 -20935.395} C_VEL
LIN {X 0,Y 209.755,Z 171.965,A -85,B 0,C 180,E1 -20936.95,E2 -20936.95} C_VEL
LIN {X 0,Y 209.438,Z 175.504,A -85,B 0,C 180,E1 -20938.296,E2 -20938.296} C_VEL
LIN {X 0,Y 209.597,Z 176.644,A -85,B 0,C 180,E1 -20938.751,E2 -20938.751} C_VEL
LIN {X 0,Y 209.735,Z 177.278,A -85,B 0,C 180,E1 -20938.913,E2 -20938.913} C_VEL
LIN {X 0,Y 213.02,Z 188.982,A -85,B 0,C 180,E1 -20939.769,E2 -20939.769} C_VEL
LIN {X 0,Y 217.001,Z 233.233,A -85,B 0,C 180,E1 -20942.208,E2 -20942.208} C_VEL
LIN {X 0,Y 214.556,Z 287.045,A -85,B 0,C 180,E1 -20944.668,E2 -20944.668} C_VEL
LIN {X 0,Y 213.421,Z 301.095,A -85,B 0,C 180,E1 -20945.694,E2 -20945.694} C_VEL
LIN {X 0,Y 211.967,Z 314.236,A -85,B 0,C 180,E1 -20947.072,E2 -20947.072} C_VEL
LIN {X 0,Y 210.497,Z 326.232,A -85,B 0,C 180,E1 -20948.736,E2 -20948.736} C_VEL
LIN {X 0,Y 208.844,Z 338.026,A -85,B 0,C 180,E1 -20950.847,E2 -20950.847} C_VEL
LIN {X 0,Y 207.362,Z 348.698,A -85,B 0,C 180,E1 -20953.257,E2 -20953.257} C_VEL
LIN {X 0,Y 206.361,Z 357.387,A -85,B 0,C 180,E1 -20955.706,E2 -20955.706} C_VEL
LIN {X 0,Y 205.466,Z 365.782,A -85,B 0,C 180,E1 -20958.658,E2 -20958.658} C_VEL
LIN {X 0,Y 205.09,Z 371.483,A -85,B 0,C 180,E1 -20961.13,E2 -20961.13} C_VEL
LIN {X 0,Y 204.97,Z 376.989,A -85,B 0,C 180,E1 -20964.097,E2 -20964.097} C_VEL
LIN {X 0,Y 204.882,Z 381.17,A -85,B 0,C 180,E1 -20967.051,E2 -20967.051} C_VEL
LIN {X 0,Y 205.029,Z 384.202,A -85,B 0,C 180,E1 -20970.001,E2 -20970.001} C_VEL
LIN {X 0,Y 204.695,Z 385.6,A -85,B 0,C 180,E1 -20971.968,E2 -20971.968} C_VEL
LIN {X 0,Y 204.496,Z 386.788,A -85,B 0,C 180,E1 -20974.679,E2 -20974.679} C_VEL
LIN {X 0,Y 204.599,Z 387.217,A -85,B 0,C 180,E1 -20977.898,E2 -20977.898} C_VEL
LIN {X 0,Y 205.461,Z 386.348,A -85,B 0,C 180,E1 -20981.844,E2 -20981.844} C_VEL
LIN {X 0,Y 206.197,Z 385.306,A -85,B 0,C 180,E1 -20983.804,E2 -20983.804} C_VEL
LIN {X 0,Y 208.697,Z 382.048,A -85,B 0,C 180,E1 -20987.643,E2 -20987.643} C_VEL
LIN {X 0,Y 211.123,Z 378.537,A -85,B 0,C 180,E1 -20990.459,E2 -20990.459} C_VEL
LIN {X 0,Y 214.015,Z 374.019,A -85,B 0,C 180,E1 -20993.208,E2 -20993.208} C_VEL
LIN {X 0,Y 217.709,Z 368.346,A -85,B 0,C 180,E1 -20995.837,E2 -20995.837} C_VEL
LIN {X 0,Y 221.878,Z 361.457,A -85,B 0,C 180,E1 -20998.368,E2 -20998.368} C_VEL
LIN {X 0,Y 226.591,Z 353.058,A -85,B 0,C 180,E1 -21000.782,E2 -21000.782} C_VEL
LIN {X 0,Y 230.955,Z 344.556,A -85,B 0,C 180,E1 -21002.693,E2 -21002.693} C_VEL
LIN {X 0,Y 236.029,Z 333.228,A -85,B 0,C 180,E1 -21004.714,E2 -21004.714} C_VEL
LIN {X 0,Y 240.592,Z 321.868,A -85,B 0,C 180,E1 -21006.266,E2 -21006.266} C_VEL
LIN {X 0,Y 244.933,Z 309.045,A -85,B 0,C 180,E1 -21007.571,E2 -21007.571} C_VEL
LIN {X 0,Y 248.345,Z 296.717,A -85,B 0,C 180,E1 -21008.506,E2 -21008.506} C_VEL
LIN {X 0,Y 251.135,Z 282.836,A -85,B 0,C 180,E1 -21009.284,E2 -21009.284} C_VEL
LIN {X 0,Y 256.022,Z 244.417,A -85,B 0,C 180,E1 -21010.81,E2 -21010.81} C_VEL
LIN {X 0,Y 255.946,Z 237.745,A -85,B 0,C 180,E1 -21011.459,E2 -21011.459} C_VEL
LIN {X 0,Y 253.463,Z 230.503,A -85,B 0,C 180,E1 -21013.289,E2 -21013.289} C_VEL
LIN {X 0,Y 250.861,Z 223.832,A -85,B 0,C 180,E1 -21015.458,E2 -21015.458} C_VEL
LIN {X 0,Y 248.934,Z 219.248,A -85,B 0,C 180,E1 -21017.345,E2 -21017.345} C_VEL
LIN {X 0,Y 246.72,Z 214.297,A -85,B 0,C 180,E1 -21020.007,E2 -21020.007} C_VEL
LIN {X 0,Y 244.547,Z 209.282,A -85,B 0,C 180,E1 -21024.257,E2 -21024.257} C_VEL
LIN {X 0,Y 244.095,Z 207.777,A -85,B 0,C 180,E1 -21026.614,E2 -21026.614} C_VEL
LIN {X 0,Y 244.207,Z 207.403,A -85,B 0,C 180,E1 -21029.698,E2 -21029.698} C_VEL
LIN {X 0,Y 245.179,Z 208.427,A -85,B 0,C 180,E1 -21032.7,E2 -21032.7} C_VEL
LIN {X 0,Y 246.808,Z 210.139,A -85,B 0,C 180,E1 -21035.328,E2 -21035.328} C_VEL
LIN {X 0,Y 249.287,Z 213.715,A -85,B 0,C 180,E1 -21038.19,E2 -21038.19} C_VEL
LIN {X 0,Y 251.769,Z 217.672,A -85,B 0,C 180,E1 -21040.428,E2 -21040.428} C_VEL
LIN {X 0,Y 254.875,Z 223.257,A -85,B 0,C 180,E1 -21042.755,E2 -21042.755} C_VEL
LIN {X 0,Y 257.601,Z 228.624,A -85,B 0,C 180,E1 -21044.507,E2 -21044.507} C_VEL
LIN {X 0,Y 252.518,Z 268.392,A -85,B 0,C 180,E1 -21046.081,E2 -21046.081} C_VEL
LIN {X 0,Y 250.129,Z 281.727,A -85,B 0,C 180,E1 -21046.896,E2 -21046.896} C_VEL
LIN {X 0,Y 247.259,Z 293.768,A -85,B 0,C 180,E1 -21047.899,E2 -21047.899} C_VEL
LIN {X 0,Y 243.553,Z 306.018,A -85,B 0,C 180,E1 -21049.268,E2 -21049.268} C_VEL
LIN {X 0,Y 239.247,Z 317.555,A -85,B 0,C 180,E1 -21050.915,E2 -21050.915} C_VEL
LIN {X 0,Y 235.051,Z 327.171,A -85,B 0,C 180,E1 -21052.699,E2 -21052.699} C_VEL
LIN {X 0,Y 230.634,Z 336.097,A -85,B 0,C 180,E1 -21054.754,E2 -21054.754} C_VEL
LIN {X 0,Y 226.507,Z 343.519,A -85,B 0,C 180,E1 -21056.919,E2 -21056.919} C_VEL
LIN {X 0,Y 222.034,Z 350.605,A -85,B 0,C 180,E1 -21059.546,E2 -21059.546} C_VEL
LIN {X 0,Y 217.289,Z 357.209,A -85,B 0,C 180,E1 -21062.861,E2 -21062.861} C_VEL
LIN {X 0,Y 213.998,Z 361.243,A -85,B 0,C 180,E1 -21065.653,E2 -21065.653} C_VEL
LIN {X 0,Y 212.027,Z 363.38,A -85,B 0,C 180,E1 -21067.618,E2 -21067.618} C_VEL
LIN {X 0,Y 210.29,Z 364.989,A -85,B 0,C 180,E1 -21069.619,E2 -21069.619} C_VEL
LIN {X 0,Y 208.488,Z 366.382,A -85,B 0,C 180,E1 -21072.155,E2 -21072.155} C_VEL
LIN {X 0,Y 206.469,Z 367.098,A -85,B 0,C 180,E1 -21075.801,E2 -21075.801} C_VEL
LIN {X 0,Y 205.649,Z 366.88,A -85,B 0,C 180,E1 -21077.912,E2 -21077.912} C_VEL
LIN {X 0,Y 205.034,Z 366.181,A -85,B 0,C 180,E1 -21080.045,E2 -21080.045} C_VEL
LIN {X 0,Y 204.597,Z 364.974,A -85,B 0,C 180,E1 -21082.2,E2 -21082.2} C_VEL
LIN {X 0,Y 204.35,Z 362.228,A -85,B 0,C 180,E1 -21085.46,E2 -21085.46} C_VEL
LIN {X 0,Y 204.569,Z 358.212,A -85,B 0,C 180,E1 -21088.748,E2 -21088.748} C_VEL
LIN {X 0,Y 205.05,Z 352.676,A -85,B 0,C 180,E1 -21092.089,E2 -21092.089} C_VEL
LIN {X 0,Y 205.812,Z 345.307,A -85,B 0,C 180,E1 -21095.486,E2 -21095.486} C_VEL
LIN {X 0,Y 206.695,Z 337.919,A -85,B 0,C 180,E1 -21098.197,E2 -21098.197} C_VEL
LIN {X 0,Y 207.938,Z 328.752,A -85,B 0,C 180,E1 -21100.907,E2 -21100.907} C_VEL
LIN {X 0,Y 209.203,Z 319.243,A -85,B 0,C 180,E1 -21103.194,E2 -21103.194} C_VEL
LIN {X 0,Y 210.679,Z 307.953,A -85,B 0,C 180,E1 -21105.39,E2 -21105.39} C_VEL
LIN {X 0,Y 212.181,Z 295.383,A -85,B 0,C 180,E1 -21107.299,E2 -21107.299} C_VEL
LIN {X 0,Y 213.353,Z 283.61,A -85,B 0,C 180,E1 -21108.688,E2 -21108.688} C_VEL
LIN {X 0,Y 214.401,Z 269.837,A -85,B 0,C 180,E1 -21109.878,E2 -21109.878} C_VEL
LIN {X 0,Y 215.166,Z 255.858,A -85,B 0,C 180,E1 -21110.687,E2 -21110.687} C_VEL
LIN {X 0,Y 218.237,Z 194.96,A -85,B 0,C 180,E1 -21113.351,E2 -21113.351} C_VEL
LIN {X 0,Y 207.468,Z 165.028,A -85,B 0,C 180,E1 -21115.724,E2 -21115.724} C_VEL
LIN {X 0,Y 206.769,Z 162.729,A -85,B 0,C 180,E1 -21115.96,E2 -21115.96} C_VEL
LIN {X 0,Y 206.724,Z 162.738,A -85,B 0,C 180,E1 -21119.338,E2 -21119.338} C_VEL
LIN {X 0,Y 206.732,Z 162.735,A -85,B 0,C 180,E1 -21123.771,E2 -21123.771} C_VEL
LIN {X 0,Y 206.754,Z 162.73,A -85,B 0,C 180,E1 -21128.042,E2 -21128.042} C_VEL
LIN {X 0,Y 206.826,Z 162.72,A -85,B 0,C 180,E1 -21132.192,E2 -21132.192} C_VEL
LIN {X 0,Y 206.881,Z 162.71,A -85,B 0,C 180,E1 -21136.243,E2 -21136.243} C_VEL
LIN {X 0,Y 207.105,Z 162.686,A -85,B 0,C 180,E1 -21140.231,E2 -21140.231} C_VEL
LIN {X 0,Y 207.166,Z 162.678,A -85,B 0,C 180,E1 -21142.2,E2 -21142.2} C_VEL
LIN {X 0,Y 207.381,Z 162.651,A -85,B 0,C 180,E1 -21148.057,E2 -21148.057} C_VEL
LIN {X 0,Y 207.514,Z 162.634,A -85,B 0,C 180,E1 -21149.999,E2 -21149.999} C_VEL
LIN {X 0,Y 207.381,Z 162.649,A -85,B 0,C 180,E1 -21151.941,E2 -21151.941} C_VEL
LIN {X 0,Y 207.166,Z 162.678,A -85,B 0,C 180,E1 -21157.798,E2 -21157.798} C_VEL
LIN {X 0,Y 206.98,Z 162.698,A -85,B 0,C 180,E1 -21161.754,E2 -21161.754} C_VEL
LIN {X 0,Y 206.865,Z 162.716,A -85,B 0,C 180,E1 -21165.77,E2 -21165.77} C_VEL
LIN {X 0,Y 206.776,Z 162.724,A -85,B 0,C 180,E1 -21169.869,E2 -21169.869} C_VEL
LIN {X 0,Y 206.745,Z 162.733,A -85,B 0,C 180,E1 -21174.074,E2 -21174.074} C_VEL
LIN {X 0,Y 206.742,Z 162.731,A -85,B 0,C 180,E1 -21178.418,E2 -21178.418} C_VEL
LIN {X 0,Y 206.707,Z 162.735,A -85,B 0,C 180,E1 -21182.955,E2 -21182.955} C_VEL
LIN {X 0,Y 206.722,Z 162.733,A -85,B 0,C 180,E1 -21187.73,E2 -21187.73} C_VEL
LIN {X 0,Y 206.72,Z 162.735,A -85,B 0,C 180,E1 -21191.588,E2 -21191.588} C_VEL
LIN {X 0,Y 206.715,Z 162.733,A -85,B 0,C 180,E1 -21195.558,E2 -21195.558} C_VEL
LIN {X 0,Y 206.717,Z 162.736,A -85,B 0,C 180,E1 -21199.763,E2 -21199.763} C_VEL
LIN {X 0,Y 206.721,Z 162.73,A -85,B 0,C 180,E1 -21202.27,E2 -21202.27} C_VEL
LIN {X 0,Y 206.706,Z 162.736,A -85,B 0,C 180,E1 -21207.045,E2 -21207.045} C_VEL
LIN {X 0,Y 206.764,Z 162.727,A -85,B 0,C 180,E1 -21212.097,E2 -21212.097} C_VEL
LIN {X 0,Y 206.783,Z 162.725,A -85,B 0,C 180,E1 -21216.584,E2 -21216.584} C_VEL
LIN {X 0,Y 206.871,Z 162.714,A -85,B 0,C 180,E1 -21222.197,E2 -21222.197} C_VEL
LIN {X 0,Y 206.912,Z 162.708,A -85,B 0,C 180,E1 -21226.246,E2 -21226.246} C_VEL
LIN {X 0,Y 207.103,Z 162.685,A -85,B 0,C 180,E1 -21230.232,E2 -21230.232} C_VEL
LIN {X 0,Y 207.165,Z 162.678,A -85,B 0,C 180,E1 -21232.202,E2 -21232.202} C_VEL
LIN {X 0,Y 207.381,Z 162.65,A -85,B 0,C 180,E1 -21238.059,E2 -21238.059} C_VEL
LIN {X 0,Y 207.514,Z 162.635,A -85,B 0,C 180,E1 -21240.001,E2 -21240.001} C_VEL
LIN {X 0,Y 207.381,Z 162.65,A -85,B 0,C 180,E1 -21241.943,E2 -21241.943} C_VEL
LIN {X 0,Y 207.188,Z 162.675,A -85,B 0,C 180,E1 -21247.799,E2 -21247.799} C_VEL
LIN {X 0,Y 206.982,Z 162.698,A -85,B 0,C 180,E1 -21251.756,E2 -21251.756} C_VEL
LIN {X 0,Y 206.866,Z 162.715,A -85,B 0,C 180,E1 -21255.772,E2 -21255.772} C_VEL
LIN {X 0,Y 206.778,Z 162.725,A -85,B 0,C 180,E1 -21259.87,E2 -21259.87} C_VEL
LIN {X 0,Y 206.746,Z 162.732,A -85,B 0,C 180,E1 -21264.075,E2 -21264.075} C_VEL
LIN {X 0,Y 206.744,Z 162.729,A -85,B 0,C 180,E1 -21268.42,E2 -21268.42} C_VEL
LIN {X 0,Y 206.709,Z 162.735,A -85,B 0,C 180,E1 -21272.957,E2 -21272.957} C_VEL
LIN {X 0,Y 206.722,Z 162.732,A -85,B 0,C 180,E1 -21275.321,E2 -21275.321} C_VEL
LIN {X 0,Y 206.679,Z 162.741,A -85,B 0,C 180,E1 -21280.248,E2 -21280.248} C_VEL
LIN {X 0,Y 206.678,Z 162.736,A -85,B 0,C 180,E1 -21284.432,E2 -21284.432} C_VEL
LIN {X 0,Y 206.664,Z 162.743,A -85,B 0,C 180,E1 -21289.75,E2 -21289.75} C_VEL
LIN {X 0,Y 206.802,Z 162.825,A -85,B 0,C 180,E1 -21293.061,E2 -21293.061} C_VEL
LIN {X 0,Y 208.935,Z 173.39,A -85,B 0,C 180,E1 -21297.44,E2 -21297.44} C_VEL
LIN {X 0,Y 209.597,Z 176.644,A -85,B 0,C 180,E1 -21298.751,E2 -21298.751} C_VEL
LIN {X 0,Y 210.407,Z 177.782,A -85,B 0,C 180,E1 -21298.997,E2 -21298.997} C_VEL
LIN {X 0,Y 214.961,Z 183.279,A -85,B 0,C 180,E1 -21299.632,E2 -21299.632} C_VEL
LIN {X 0,Y 216.352,Z 187.099,A -85,B 0,C 180,E1 -21299.948,E2 -21299.948} C_VEL
LIN {X 0,Y 216.283,Z 189.984,A -85,B 0,C 180,E1 -21300.05,E2 -21300.05} C_VEL
LIN {X 0,Y 214.477,Z 194.168,A -85,B 0,C 180,E1 -21300.111,E2 -21300.111} C_VEL
LIN {X 0,Y 210.795,Z 200.373,A -85,B 0,C 180,E1 -21300.149,E2 -21300.149} C_VEL
LIN {X 0,Y 209.89,Z 203.602,A -85,B 0,C 180,E1 -21300.233,E2 -21300.233} C_VEL
LIN {X 0,Y 208.817,Z 204.167,A -85,B 0,C 180,E1 -21300.179,E2 -21300.179} C_VEL
LIN {X 0,Y 207.716,Z 207.866,A -85,B 0,C 180,E1 -21300.275,E2 -21300.275} C_VEL
LIN {X 0,Y 210.087,Z 234.447,A -85,B 0,C 180,E1 -21301.78,E2 -21301.78} C_VEL
LIN {X 0,Y 207.648,Z 286.324,A -85,B 0,C 180,E1 -21304.234,E2 -21304.234} C_VEL
LIN {X 0,Y 206.555,Z 299.699,A -85,B 0,C 180,E1 -21305.234,E2 -21305.234} C_VEL
LIN {X 0,Y 205.188,Z 312.142,A -85,B 0,C 180,E1 -21306.537,E2 -21306.537} C_VEL
LIN {X 0,Y 203.683,Z 324.246,A -85,B 0,C 180,E1 -21308.229,E2 -21308.229} C_VEL
LIN {X 0,Y 202.14,Z 335.314,A -85,B 0,C 180,E1 -21310.192,E2 -21310.192} C_VEL
LIN {X 0,Y 200.527,Z 346.314,A -85,B 0,C 180,E1 -21312.669,E2 -21312.669} C_VEL
LIN {X 0,Y 199.472,Z 355.356,A -85,B 0,C 180,E1 -21315.201,E2 -21315.201} C_VEL
LIN {X 0,Y 198.636,Z 362.782,A -85,B 0,C 180,E1 -21317.744,E2 -21317.744} C_VEL
LIN {X 0,Y 198.09,Z 370.042,A -85,B 0,C 180,E1 -21320.814,E2 -21320.814} C_VEL
LIN {X 0,Y 197.912,Z 375.753,A -85,B 0,C 180,E1 -21323.885,E2 -21323.885} C_VEL
LIN {X 0,Y 197.853,Z 380.134,A -85,B 0,C 180,E1 -21326.946,E2 -21326.946} C_VEL
LIN {X 0,Y 197.973,Z 383.342,A -85,B 0,C 180,E1 -21330.001,E2 -21330.001} C_VEL
LIN {X 0,Y 197.544,Z 385.884,A -85,B 0,C 180,E1 -21334.081,E2 -21334.081} C_VEL
LIN {X 0,Y 197.419,Z 386.529,A -85,B 0,C 180,E1 -21336.132,E2 -21336.132} C_VEL
LIN {X 0,Y 197.919,Z 386.605,A -85,B 0,C 180,E1 -21340.228,E2 -21340.228} C_VEL
LIN {X 0,Y 199.276,Z 385.167,A -85,B 0,C 180,E1 -21344.293,E2 -21344.293} C_VEL
LIN {X 0,Y 200.46,Z 383.881,A -85,B 0,C 180,E1 -21346.289,E2 -21346.289} C_VEL
LIN {X 0,Y 203.57,Z 380.058,A -85,B 0,C 180,E1 -21350.197,E2 -21350.197} C_VEL
LIN {X 0,Y 207.071,Z 375.206,A -85,B 0,C 180,E1 -21353.596,E2 -21353.596} C_VEL
LIN {X 0,Y 211.412,Z 369.204,A -85,B 0,C 180,E1 -21356.666,E2 -21356.666} C_VEL
LIN {X 0,Y 216.49,Z 361.349,A -85,B 0,C 180,E1 -21359.675,E2 -21359.675} C_VEL
LIN {X 0,Y 221.51,Z 353.007,A -85,B 0,C 180,E1 -21362.103,E2 -21362.103} C_VEL
LIN {X 0,Y 226.1,Z 344.701,A -85,B 0,C 180,E1 -21364.022,E2 -21364.022} C_VEL
LIN {X 0,Y 231.421,Z 333.614,A -85,B 0,C 180,E1 -21366.044,E2 -21366.044} C_VEL
LIN {X 0,Y 236.166,Z 322.41,A -85,B 0,C 180,E1 -21367.594,E2 -21367.594} C_VEL
LIN {X 0,Y 240.672,Z 309.899,A -85,B 0,C 180,E1 -21368.891,E2 -21368.891} C_VEL
LIN {X 0,Y 244.509,Z 296.959,A -85,B 0,C 180,E1 -21369.892,E2 -21369.892} C_VEL
LIN {X 0,Y 247.419,Z 283.693,A -85,B 0,C 180,E1 -21370.659,E2 -21370.659} C_VEL
LIN {X 0,Y 250.228,Z 263.887,A -85,B 0,C 180,E1 -21371.473,E2 -21371.473} C_VEL
LIN {X 0,Y 252.546,Z 245.579,A -85,B 0,C 180,E1 -21372.205,E2 -21372.205} C_VEL
LIN {X 0,Y 252.499,Z 241.611,A -85,B 0,C 180,E1 -21372.614,E2 -21372.614} C_VEL
LIN {X 0,Y 250.298,Z 234.534,A -85,B 0,C 180,E1 -21374.519,E2 -21374.519} C_VEL
LIN {X 0,Y 248.227,Z 229.151,A -85,B 0,C 180,E1 -21376.42,E2 -21376.42} C_VEL
LIN {X 0,Y 246.769,Z 225.387,A -85,B 0,C 180,E1 -21378.014,E2 -21378.014} C_VEL
LIN {X 0,Y 244.924,Z 220.849,A -85,B 0,C 180,E1 -21380.491,E2 -21380.491} C_VEL
LIN {X 0,Y 242.923,Z 215.783,A -85,B 0,C 180,E1 -21384.941,E2 -21384.941} C_VEL
LIN {X 0,Y 242.657,Z 214.603,A -85,B 0,C 180,E1 -21387.132,E2 -21387.132} C_VEL
LIN {X 0,Y 242.924,Z 214.442,A -85,B 0,C 180,E1 -21390.22,E2 -21390.22} C_VEL
LIN {X 0,Y 244.327,Z 216.077,A -85,B 0,C 180,E1 -21393.797,E2 -21393.797} C_VEL
LIN {X 0,Y 245.343,Z 217.217,A -85,B 0,C 180,E1 -21395.289,E2 -21395.289} C_VEL
LIN {X 0,Y 247.377,Z 220.313,A -85,B 0,C 180,E1 -21397.768,E2 -21397.768} C_VEL
LIN {X 0,Y 249.575,Z 224.004,A -85,B 0,C 180,E1 -21399.885,E2 -21399.885} C_VEL
LIN {X 0,Y 252.346,Z 229.211,A -85,B 0,C 180,E1 -21402.095,E2 -21402.095} C_VEL
LIN {X 0,Y 253.87,Z 232.426,A -85,B 0,C 180,E1 -21403.217,E2 -21403.217} C_VEL
LIN {X 0,Y 248.84,Z 270.168,A -85,B 0,C 180,E1 -21404.738,E2 -21404.738} C_VEL
LIN {X 0,Y 246.359,Z 283.006,A -85,B 0,C 180,E1 -21405.544,E2 -21405.544} C_VEL
LIN {X 0,Y 243.077,Z 295.571,A -85,B 0,C 180,E1 -21406.626,E2 -21406.626} C_VEL
LIN {X 0,Y 239.356,Z 306.947,A -85,B 0,C 180,E1 -21407.924,E2 -21407.924} C_VEL
LIN {X 0,Y 235.423,Z 317.059,A -85,B 0,C 180,E1 -21409.352,E2 -21409.352} C_VEL
LIN {X 0,Y 231.227,Z 326.441,A -85,B 0,C 180,E1 -21411.038,E2 -21411.038} C_VEL
LIN {X 0,Y 226.552,Z 335.42,A -85,B 0,C 180,E1 -21413.072,E2 -21413.072} C_VEL
LIN {X 0,Y 221.645,Z 343.675,A -85,B 0,C 180,E1 -21415.453,E2 -21415.453} C_VEL
LIN {X 0,Y 216.83,Z 350.927,A -85,B 0,C 180,E1 -21418.142,E2 -21418.142} C_VEL
LIN {X 0,Y 212.522,Z 356.599,A -85,B 0,C 180,E1 -21420.947,E2 -21420.947} C_VEL
LIN {X 0,Y 208.708,Z 360.973,A -85,B 0,C 180,E1 -21423.861,E2 -21423.861} C_VEL
LIN {X 0,Y 205.349,Z 364.314,A -85,B 0,C 180,E1 -21427.009,E2 -21427.009} C_VEL
LIN {X 0,Y 202.841,Z 366.321,A -85,B 0,C 180,E1 -21429.975,E2 -21429.975} C_VEL
LIN {X 0,Y 201.307,Z 367.184,A -85,B 0,C 180,E1 -21432.166,E2 -21432.166} C_VEL
LIN {X 0,Y 200.13,Z 367.556,A -85,B 0,C 180,E1 -21434.23,E2 -21434.23} C_VEL
LIN {X 0,Y 198.744,Z 367.304,A -85,B 0,C 180,E1 -21437.295,E2 -21437.295} C_VEL
LIN {X 0,Y 197.741,Z 365.886,A -85,B 0,C 180,E1 -21440.818,E2 -21440.818} C_VEL
LIN {X 0,Y 197.294,Z 363.384,A -85,B 0,C 180,E1 -21444.182,E2 -21444.182} C_VEL
LIN {X 0,Y 197.336,Z 359.661,A -85,B 0,C 180,E1 -21447.579,E2 -21447.579} C_VEL
LIN {X 0,Y 197.697,Z 355.098,A -85,B 0,C 180,E1 -21450.684,E2 -21450.684} C_VEL
LIN {X 0,Y 198.308,Z 348.939,A -85,B 0,C 180,E1 -21453.929,E2 -21453.929} C_VEL
LIN {X 0,Y 199.133,Z 341.932,A -85,B 0,C 180,E1 -21456.868,E2 -21456.868} C_VEL
LIN {X 0,Y 200.234,Z 333.3,A -85,B 0,C 180,E1 -21459.773,E2 -21459.773} C_VEL
LIN {X 0,Y 201.682,Z 322.738,A -85,B 0,C 180,E1 -21462.62,E2 -21462.62} C_VEL
LIN {X 0,Y 203.076,Z 312.437,A -85,B 0,C 180,E1 -21464.839,E2 -21464.839} C_VEL
LIN {X 0,Y 204.623,Z 300.167,A -85,B 0,C 180,E1 -21466.943,E2 -21466.943} C_VEL
LIN {X 0,Y 205.886,Z 288.637,A -85,B 0,C 180,E1 -21468.495,E2 -21468.495} C_VEL
LIN {X 0,Y 207.138,Z 275.087,A -85,B 0,C 180,E1 -21469.86,E2 -21469.86} C_VEL
LIN {X 0,Y 207.973,Z 261.876,A -85,B 0,C 180,E1 -21470.804,E2 -21470.804} C_VEL
LIN {X 0,Y 211.279,Z 196.008,A -85,B 0,C 180,E1 -21473.856,E2 -21473.856} C_VEL
LIN {X 0,Y 200.262,Z 165.622,A -85,B 0,C 180,E1 -21476.345,E2 -21476.345} C_VEL
LIN {X 0,Y 199.682,Z 163.611,A -85,B 0,C 180,E1 -21476.523,E2 -21476.523} C_VEL
LIN {X 0,Y 199.712,Z 163.612,A -85,B 0,C 180,E1 -21481.612,E2 -21481.612} C_VEL
LIN {X 0,Y 199.736,Z 163.607,A -85,B 0,C 180,E1 -21487.228,E2 -21487.228} C_VEL
LIN {X 0,Y 199.75,Z 163.602,A -85,B 0,C 180,E1 -21491.797,E2 -21491.797} C_VEL
LIN {X 0,Y 199.818,Z 163.59,A -85,B 0,C 180,E1 -21495.746,E2 -21495.746} C_VEL
LIN {X 0,Y 200.069,Z 163.562,A -85,B 0,C 180,E1 -21499.883,E2 -21499.883} C_VEL
LIN {X 0,Y 200.033,Z 163.564,A -85,B 0,C 180,E1 -21503.949,E2 -21503.949} C_VEL
LIN {X 0,Y 200.321,Z 163.53,A -85,B 0,C 180,E1 -21507.989,E2 -21507.989} C_VEL
LIN {X 0,Y 200.479,Z 163.511,A -85,B 0,C 180,E1 -21509.999,E2 -21509.999} C_VEL
LIN {X 0,Y 200.029,Z 163.564,A -85,B 0,C 180,E1 -21514.029,E2 -21514.029} C_VEL
LIN {X 0,Y 200.109,Z 163.558,A -85,B 0,C 180,E1 -21518.075,E2 -21518.075} C_VEL
LIN {X 0,Y 199.912,Z 163.579,A -85,B 0,C 180,E1 -21522.176,E2 -21522.176} C_VEL
LIN {X 0,Y 199.803,Z 163.598,A -85,B 0,C 180,E1 -21526.343,E2 -21526.343} C_VEL
LIN {X 0,Y 199.688,Z 163.61,A -85,B 0,C 180,E1 -21530.606,E2 -21530.606} C_VEL
LIN {X 0,Y 199.662,Z 163.612,A -85,B 0,C 180,E1 -21534.985,E2 -21534.985} C_VEL
LIN {X 0,Y 199.672,Z 163.61,A -85,B 0,C 180,E1 -21539.522,E2 -21539.522} C_VEL
LIN {X 0,Y 199.662,Z 163.614,A -85,B 0,C 180,E1 -21542.352,E2 -21542.352} C_VEL
LIN {X 0,Y 199.65,Z 163.612,A -85,B 0,C 180,E1 -21546.756,E2 -21546.756} C_VEL
LIN {X 0,Y 199.675,Z 163.611,A -85,B 0,C 180,E1 -21549.311,E2 -21549.311} C_VEL
LIN {X 0,Y 199.659,Z 163.612,A -85,B 0,C 180,E1 -21552.338,E2 -21552.338} C_VEL
LIN {X 0,Y 199.662,Z 163.61,A -85,B 0,C 180,E1 -21555.253,E2 -21555.253} C_VEL
LIN {X 0,Y 199.659,Z 163.615,A -85,B 0,C 180,E1 -21558.027,E2 -21558.027} C_VEL
LIN {X 0,Y 199.676,Z 163.61,A -85,B 0,C 180,E1 -21560.743,E2 -21560.743} C_VEL
LIN {X 0,Y 199.632,Z 163.619,A -85,B 0,C 180,E1 -21565.718,E2 -21565.718} C_VEL
LIN {X 0,Y 199.701,Z 163.608,A -85,B 0,C 180,E1 -21568.138,E2 -21568.138} C_VEL
LIN {X 0,Y 199.684,Z 163.608,A -85,B 0,C 180,E1 -21572.772,E2 -21572.772} C_VEL
LIN {X 0,Y 199.735,Z 163.606,A -85,B 0,C 180,E1 -21577.23,E2 -21577.23} C_VEL
LIN {X 0,Y 199.794,Z 163.597,A -85,B 0,C 180,E1 -21581.758,E2 -21581.758} C_VEL
LIN {X 0,Y 199.846,Z 163.588,A -85,B 0,C 180,E1 -21585.75,E2 -21585.75} C_VEL
LIN {X 0,Y 200.068,Z 163.562,A -85,B 0,C 180,E1 -21589.885,E2 -21589.885} C_VEL
LIN {X 0,Y 200.032,Z 163.565,A -85,B 0,C 180,E1 -21593.95,E2 -21593.95} C_VEL
LIN {X 0,Y 200.32,Z 163.53,A -85,B 0,C 180,E1 -21597.99,E2 -21597.99} C_VEL
LIN {X 0,Y 200.478,Z 163.511,A -85,B 0,C 180,E1 -21600.001,E2 -21600.001} C_VEL
LIN {X 0,Y 200.031,Z 163.563,A -85,B 0,C 180,E1 -21604.03,E2 -21604.03} C_VEL
LIN {X 0,Y 200.131,Z 163.555,A -85,B 0,C 180,E1 -21608.076,E2 -21608.076} C_VEL
LIN {X 0,Y 199.914,Z 163.58,A -85,B 0,C 180,E1 -21612.178,E2 -21612.178} C_VEL
LIN {X 0,Y 199.804,Z 163.597,A -85,B 0,C 180,E1 -21616.344,E2 -21616.344} C_VEL
LIN {X 0,Y 199.69,Z 163.608,A -85,B 0,C 180,E1 -21620.607,E2 -21620.607} C_VEL
LIN {X 0,Y 199.664,Z 163.613,A -85,B 0,C 180,E1 -21624.986,E2 -21624.986} C_VEL
LIN {X 0,Y 199.675,Z 163.608,A -85,B 0,C 180,E1 -21629.523,E2 -21629.523} C_VEL
LIN {X 0,Y 199.665,Z 163.615,A -85,B 0,C 180,E1 -21632.354,E2 -21632.354} C_VEL
LIN {X 0,Y 199.64,Z 163.612,A -85,B 0,C 180,E1 -21636.76,E2 -21636.76} C_VEL
LIN {X 0,Y 199.641,Z 163.614,A -85,B 0,C 180,E1 -21639.321,E2 -21639.321} C_VEL
LIN {X 0,Y 199.62,Z 163.619,A -85,B 0,C 180,E1 -21642.326,E2 -21642.326} C_VEL
LIN {X 0,Y 199.595,Z 163.618,A -85,B 0,C 180,E1 -21645.234,E2 -21645.234} C_VEL
LIN {X 0,Y 199.641,Z 163.615,A -85,B 0,C 180,E1 -21650.758,E2 -21650.758} C_VEL
LIN {X 0,Y 199.732,Z 163.688,A -85,B 0,C 180,E1 -21652.709,E2 -21652.709} C_VEL
LIN {X 0,Y 201.913,Z 174.527,A -85,B 0,C 180,E1 -21657.352,E2 -21657.352} C_VEL
LIN {X 0,Y 202.395,Z 176.796,A -85,B 0,C 180,E1 -21658.237,E2 -21658.237} C_VEL
LIN {X 0,Y 206.263,Z 190.217,A -85,B 0,C 180,E1 -21659.264,E2 -21659.264} C_VEL
LIN {X 0,Y 207.716,Z 207.866,A -85,B 0,C 180,E1 -21660.275,E2 -21660.275} C_VEL
LIN {X 0,Y 207.65,Z 213.678,A -85,B 0,C 180,E1 -21660.56,E2 -21660.56} C_VEL
LIN {X 0,Y 205.889,Z 223.33,A -85,B 0,C 180,E1 -21660.918,E2 -21660.918} C_VEL
LIN {X 0,Y 203.384,Z 234.954,A -85,B 0,C 180,E1 -21661.333,E2 -21661.333} C_VEL
LIN {X 0,Y 203,Z 238.871,A -85,B 0,C 180,E1 -21661.508,E2 -21661.508} C_VEL
LIN {X 0,Y 200.644,Z 286.79,A -85,B 0,C 180,E1 -21663.895,E2 -21663.895} C_VEL
LIN {X 0,Y 199.487,Z 300.599,A -85,B 0,C 180,E1 -21664.992,E2 -21664.992} C_VEL
LIN {X 0,Y 197.971,Z 313.579,A -85,B 0,C 180,E1 -21666.462,E2 -21666.462} C_VEL
LIN {X 0,Y 196.461,Z 325.348,A -85,B 0,C 180,E1 -21668.216,E2 -21668.216} C_VEL
LIN {X 0,Y 194.879,Z 336.494,A -85,B 0,C 180,E1 -21670.338,E2 -21670.338} C_VEL
LIN {X 0,Y 193.45,Z 345.886,A -85,B 0,C 180,E1 -21672.56,E2 -21672.56} C_VEL
LIN {X 0,Y 192.381,Z 354.935,A -85,B 0,C 180,E1 -21675.185,E2 -21675.185} C_VEL
LIN {X 0,Y 191.559,Z 362.369,A -85,B 0,C 180,E1 -21677.822,E2 -21677.822} C_VEL
LIN {X 0,Y 191.026,Z 369.63,A -85,B 0,C 180,E1 -21681.005,E2 -21681.005} C_VEL
LIN {X 0,Y 190.887,Z 375.983,A -85,B 0,C 180,E1 -21684.612,E2 -21684.612} C_VEL
LIN {X 0,Y 190.778,Z 380.279,A -85,B 0,C 180,E1 -21687.89,E2 -21687.89} C_VEL
LIN {X 0,Y 190.938,Z 382.432,A -85,B 0,C 180,E1 -21690.001,E2 -21690.001} C_VEL
LIN {X 0,Y 190.581,Z 383.998,A -85,B 0,C 180,E1 -21692.114,E2 -21692.114} C_VEL
LIN {X 0,Y 190.386,Z 385.333,A -85,B 0,C 180,E1 -21694.653,E2 -21694.653} C_VEL
LIN {X 0,Y 190.499,Z 386.268,A -85,B 0,C 180,E1 -21698.487,E2 -21698.487} C_VEL
LIN {X 0,Y 190.92,Z 386.236,A -85,B 0,C 180,E1 -21700.607,E2 -21700.607} C_VEL
LIN {X 0,Y 192.371,Z 384.997,A -85,B 0,C 180,E1 -21704.818,E2 -21704.818} C_VEL
LIN {X 0,Y 195.179,Z 382.263,A -85,B 0,C 180,E1 -21708.91,E2 -21708.91} C_VEL
LIN {X 0,Y 197.861,Z 379.152,A -85,B 0,C 180,E1 -21711.899,E2 -21711.899} C_VEL
LIN {X 0,Y 201.102,Z 375.101,A -85,B 0,C 180,E1 -21714.795,E2 -21714.795} C_VEL
LIN {X 0,Y 205.13,Z 369.974,A -85,B 0,C 180,E1 -21717.551,E2 -21717.551} C_VEL
LIN {X 0,Y 210.456,Z 362.537,A -85,B 0,C 180,E1 -21720.615,E2 -21720.615} C_VEL
LIN {X 0,Y 215.644,Z 354.618,A -85,B 0,C 180,E1 -21723.087,E2 -21723.087} C_VEL
LIN {X 0,Y 221.376,Z 344.919,A -85,B 0,C 180,E1 -21725.408,E2 -21725.408} C_VEL
LIN {X 0,Y 226.928,Z 334.05,A -85,B 0,C 180,E1 -21727.431,E2 -21727.431} C_VEL
LIN {X 0,Y 231.903,Z 323.145,A -85,B 0,C 180,E1 -21728.966,E2 -21728.966} C_VEL
LIN {X 0,Y 236.576,Z 311.161,A -85,B 0,C 180,E1 -21730.251,E2 -21730.251} C_VEL
LIN {X 0,Y 240.53,Z 298.65,A -85,B 0,C 180,E1 -21731.243,E2 -21731.243} C_VEL
LIN {X 0,Y 243.845,Z 284.779,A -85,B 0,C 180,E1 -21732.076,E2 -21732.076} C_VEL
LIN {X 0,Y 246.444,Z 268.379,A -85,B 0,C 180,E1 -21732.755,E2 -21732.755} C_VEL
LIN {X 0,Y 249.29,Z 247.293,A -85,B 0,C 180,E1 -21733.603,E2 -21733.603} C_VEL
LIN {X 0,Y 249.243,Z 245.402,A -85,B 0,C 180,E1 -21733.841,E2 -21733.841} C_VEL
LIN {X 0,Y 247.195,Z 238.857,A -85,B 0,C 180,E1 -21735.772,E2 -21735.772} C_VEL
LIN {X 0,Y 245.789,Z 234.62,A -85,B 0,C 180,E1 -21737.345,E2 -21737.345} C_VEL
LIN {X 0,Y 244.673,Z 231.639,A -85,B 0,C 180,E1 -21738.65,E2 -21738.65} C_VEL
LIN {X 0,Y 243.119,Z 227.333,A -85,B 0,C 180,E1 -21741.027,E2 -21741.027} C_VEL
LIN {X 0,Y 241.455,Z 222.424,A -85,B 0,C 180,E1 -21745.447,E2 -21745.447} C_VEL
LIN {X 0,Y 241.231,Z 221.471,A -85,B 0,C 180,E1 -21747.661,E2 -21747.661} C_VEL
LIN {X 0,Y 241.704,Z 221.6,A -85,B 0,C 180,E1 -21750.984,E2 -21750.984} C_VEL
LIN {X 0,Y 243.588,Z 223.825,A -85,B 0,C 180,E1 -21754.824,E2 -21754.824} C_VEL
LIN {X 0,Y 245.586,Z 227.102,A -85,B 0,C 180,E1 -21757.455,E2 -21757.455} C_VEL
LIN {X 0,Y 247.544,Z 230.547,A -85,B 0,C 180,E1 -21759.425,E2 -21759.425} C_VEL
LIN {X 0,Y 249.962,Z 235.375,A -85,B 0,C 180,E1 -21761.507,E2 -21761.507} C_VEL
LIN {X 0,Y 250.431,Z 236.622,A -85,B 0,C 180,E1 -21761.908,E2 -21761.908} C_VEL
LIN {X 0,Y 245.611,Z 270.396,A -85,B 0,C 180,E1 -21763.272,E2 -21763.272} C_VEL
LIN {X 0,Y 243.041,Z 283.04,A -85,B 0,C 180,E1 -21764.051,E2 -21764.051} C_VEL
LIN {X 0,Y 239.63,Z 295.76,A -85,B 0,C 180,E1 -21765.129,E2 -21765.129} C_VEL
LIN {X 0,Y 235.162,Z 308.733,A -85,B 0,C 180,E1 -21766.607,E2 -21766.607} C_VEL
LIN {X 0,Y 230.475,Z 319.706,A -85,B 0,C 180,E1 -21768.231,E2 -21768.231} C_VEL
LIN {X 0,Y 225.575,Z 329.593,A -85,B 0,C 180,E1 -21770.133,E2 -21770.133} C_VEL
LIN {X 0,Y 220.466,Z 338.598,A -85,B 0,C 180,E1 -21772.31,E2 -21772.31} C_VEL
LIN {X 0,Y 215.222,Z 346.61,A -85,B 0,C 180,E1 -21774.847,E2 -21774.847} C_VEL
LIN {X 0,Y 210.521,Z 352.859,A -85,B 0,C 180,E1 -21777.398,E2 -21777.398} C_VEL
LIN {X 0,Y 206.447,Z 357.778,A -85,B 0,C 180,E1 -21779.999,E2 -21779.999} C_VEL
LIN {X 0,Y 202.413,Z 362,A -85,B 0,C 180,E1 -21782.985,E2 -21782.985} C_VEL
LIN {X 0,Y 198.215,Z 365.646,A -85,B 0,C 180,E1 -21786.884,E2 -21786.884} C_VEL
LIN {X 0,Y 195.344,Z 367.43,A -85,B 0,C 180,E1 -21790.362,E2 -21790.362} C_VEL
LIN {X 0,Y 193.894,Z 367.938,A -85,B 0,C 180,E1 -21792.56,E2 -21792.56} C_VEL
LIN {X 0,Y 192.687,Z 368.013,A -85,B 0,C 180,E1 -21794.791,E2 -21794.791} C_VEL
LIN {X 0,Y 191.568,Z 367.451,A -85,B 0,C 180,E1 -21797.471,E2 -21797.471} C_VEL
LIN {X 0,Y 190.481,Z 365.355,A -85,B 0,C 180,E1 -21801.651,E2 -21801.651} C_VEL
LIN {X 0,Y 190.172,Z 362.318,A -85,B 0,C 180,E1 -21805.149,E2 -21805.149} C_VEL
LIN {X 0,Y 190.364,Z 357.996,A -85,B 0,C 180,E1 -21808.681,E2 -21808.681} C_VEL
LIN {X 0,Y 190.852,Z 352.433,A -85,B 0,C 180,E1 -21812.116,E2 -21812.116} C_VEL
LIN {X 0,Y 191.563,Z 345.891,A -85,B 0,C 180,E1 -21815.297,E2 -21815.297} C_VEL
LIN {X 0,Y 192.531,Z 338.047,A -85,B 0,C 180,E1 -21818.356,E2 -21818.356} C_VEL
LIN {X 0,Y 193.906,Z 328.204,A -85,B 0,C 180,E1 -21821.41,E2 -21821.41} C_VEL
LIN {X 0,Y 195.264,Z 317.985,A -85,B 0,C 180,E1 -21823.957,E2 -21823.957} C_VEL
LIN {X 0,Y 196.896,Z 306.173,A -85,B 0,C 180,E1 -21826.285,E2 -21826.285} C_VEL
LIN {X 0,Y 198.303,Z 294.621,A -85,B 0,C 180,E1 -21828.094,E2 -21828.094} C_VEL
LIN {X 0,Y 199.606,Z 282.19,A -85,B 0,C 180,E1 -21829.587,E2 -21829.587} C_VEL
LIN {X 0,Y 200.652,Z 268.077,A -85,B 0,C 180,E1 -21830.834,E2 -21830.834} C_VEL
LIN {X 0,Y 201.633,Z 250.679,A -85,B 0,C 180,E1 -21831.792,E2 -21831.792} C_VEL
LIN {X 0,Y 204.446,Z 197.513,A -85,B 0,C 180,E1 -21834.315,E2 -21834.315} C_VEL
LIN {X 0,Y 193.828,Z 168.223,A -85,B 0,C 180,E1 -21836.818,E2 -21836.818} C_VEL
LIN {X 0,Y 192.665,Z 164.486,A -85,B 0,C 180,E1 -21837.179,E2 -21837.179} C_VEL
LIN {X 0,Y 192.665,Z 164.49,A -85,B 0,C 180,E1 -21841.691,E2 -21841.691} C_VEL
LIN {X 0,Y 192.705,Z 164.481,A -85,B 0,C 180,E1 -21846.348,E2 -21846.348} C_VEL
LIN {X 0,Y 192.698,Z 164.482,A -85,B 0,C 180,E1 -21851.486,E2 -21851.486} C_VEL
LIN {X 0,Y 192.742,Z 164.474,A -85,B 0,C 180,E1 -21855.211,E2 -21855.211} C_VEL
LIN {X 0,Y 192.98,Z 164.446,A -85,B 0,C 180,E1 -21859.508,E2 -21859.508} C_VEL
LIN {X 0,Y 193.061,Z 164.435,A -85,B 0,C 180,E1 -21861.627,E2 -21861.627} C_VEL
LIN {X 0,Y 193.263,Z 164.41,A -85,B 0,C 180,E1 -21867.915,E2 -21867.915} C_VEL
LIN {X 0,Y 193.442,Z 164.387,A -85,B 0,C 180,E1 -21869.999,E2 -21869.999} C_VEL
LIN {X 0,Y 192.976,Z 164.443,A -85,B 0,C 180,E1 -21874.176,E2 -21874.176} C_VEL
LIN {X 0,Y 193.06,Z 164.437,A -85,B 0,C 180,E1 -21878.372,E2 -21878.372} C_VEL
LIN {X 0,Y 192.851,Z 164.461,A -85,B 0,C 180,E1 -21882.629,E2 -21882.629} C_VEL
LIN {X 0,Y 192.755,Z 164.473,A -85,B 0,C 180,E1 -21886.958,E2 -21886.958} C_VEL
LIN {X 0,Y 192.619,Z 164.489,A -85,B 0,C 180,E1 -21891.398,E2 -21891.398} C_VEL
LIN {X 0,Y 192.645,Z 164.49,A -85,B 0,C 180,E1 -21894.213,E2 -21894.213} C_VEL
LIN {X 0,Y 192.647,Z 164.485,A -85,B 0,C 180,E1 -21898.892,E2 -21898.892} C_VEL
LIN {X 0,Y 192.598,Z 164.492,A -85,B 0,C 180,E1 -21903.185,E2 -21903.185} C_VEL
LIN {X 0,Y 192.597,Z 164.494,A -85,B 0,C 180,E1 -21908.34,E2 -21908.34} C_VEL
LIN {X 0,Y 192.601,Z 164.491,A -85,B 0,C 180,E1 -21913.132,E2 -21913.132} C_VEL
LIN {X 0,Y 192.6,Z 164.492,A -85,B 0,C 180,E1 -21916.869,E2 -21916.869} C_VEL
LIN {X 0,Y 192.597,Z 164.492,A -85,B 0,C 180,E1 -21921.66,E2 -21921.66} C_VEL
LIN {X 0,Y 192.598,Z 164.493,A -85,B 0,C 180,E1 -21926.815,E2 -21926.815} C_VEL
LIN {X 0,Y 192.662,Z 164.484,A -85,B 0,C 180,E1 -21931.692,E2 -21931.692} C_VEL
LIN {X 0,Y 192.703,Z 164.479,A -85,B 0,C 180,E1 -21936.349,E2 -21936.349} C_VEL
LIN {X 0,Y 192.729,Z 164.478,A -85,B 0,C 180,E1 -21941.458,E2 -21941.458} C_VEL
LIN {X 0,Y 192.77,Z 164.473,A -85,B 0,C 180,E1 -21945.215,E2 -21945.215} C_VEL
LIN {X 0,Y 192.979,Z 164.446,A -85,B 0,C 180,E1 -21949.509,E2 -21949.509} C_VEL
LIN {X 0,Y 193.06,Z 164.436,A -85,B 0,C 180,E1 -21951.628,E2 -21951.628} C_VEL
LIN {X 0,Y 193.262,Z 164.409,A -85,B 0,C 180,E1 -21957.917,E2 -21957.917} C_VEL
LIN {X 0,Y 193.442,Z 164.388,A -85,B 0,C 180,E1 -21960.001,E2 -21960.001} C_VEL
LIN {X 0,Y 192.978,Z 164.442,A -85,B 0,C 180,E1 -21964.178,E2 -21964.178} C_VEL
LIN {X 0,Y 193.078,Z 164.434,A -85,B 0,C 180,E1 -21968.373,E2 -21968.373} C_VEL
LIN {X 0,Y 192.852,Z 164.46,A -85,B 0,C 180,E1 -21972.631,E2 -21972.631} C_VEL
LIN {X 0,Y 192.757,Z 164.474,A -85,B 0,C 180,E1 -21976.96,E2 -21976.96} C_VEL
LIN {X 0,Y 192.621,Z 164.487,A -85,B 0,C 180,E1 -21981.4,E2 -21981.4} C_VEL
LIN {X 0,Y 192.647,Z 164.489,A -85,B 0,C 180,E1 -21984.214,E2 -21984.214} C_VEL
LIN {X 0,Y 192.65,Z 164.483,A -85,B 0,C 180,E1 -21988.893,E2 -21988.893} C_VEL
LIN {X 0,Y 192.601,Z 164.492,A -85,B 0,C 180,E1 -21993.186,E2 -21993.186} C_VEL
LIN {X 0,Y 192.61,Z 164.488,A -85,B 0,C 180,E1 -21996.609,E2 -21996.609} C_VEL
LIN {X 0,Y 192.548,Z 164.499,A -85,B 0,C 180,E1 -22001.072,E2 -22001.072} C_VEL
LIN {X 0,Y 192.522,Z 164.504,A -85,B 0,C 180,E1 -22006.086,E2 -22006.086} C_VEL
LIN {X 0,Y 192.616,Z 164.493,A -85,B 0,C 180,E1 -22011.665,E2 -22011.665} C_VEL
LIN {X 0,Y 192.671,Z 164.608,A -85,B 0,C 180,E1 -22012.374,E2 -22012.374} C_VEL
LIN {X 0,Y 194.722,Z 174.629,A -85,B 0,C 180,E1 -22016.834,E2 -22016.834} C_VEL
LIN {X 0,Y 195.048,Z 176.372,A -85,B 0,C 180,E1 -22017.541,E2 -22017.541} C_VEL
LIN {X 0,Y 199.545,Z 191.968,A -85,B 0,C 180,E1 -22018.792,E2 -22018.792} C_VEL
LIN {X 0,Y 203.206,Z 235.004,A -85,B 0,C 180,E1 -22021.324,E2 -22021.324} C_VEL
LIN {X 0,Y 203,Z 238.871,A -85,B 0,C 180,E1 -22021.508,E2 -22021.508} C_VEL
LIN {X 0,Y 202.083,Z 244.65,A -85,B 0,C 180,E1 -22021.742,E2 -22021.742} C_VEL
LIN {X 0,Y 195.567,Z 263.309,A -85,B 0,C 180,E1 -22022.282,E2 -22022.282} C_VEL
LIN {X 0,Y 194.6,Z 269.087,A -85,B 0,C 180,E1 -22022.53,E2 -22022.53} C_VEL
LIN {X 0,Y 193.541,Z 289.114,A -85,B 0,C 180,E1 -22023.661,E2 -22023.661} C_VEL
LIN {X 0,Y 192.255,Z 302.536,A -85,B 0,C 180,E1 -22024.853,E2 -22024.853} C_VEL
LIN {X 0,Y 190.756,Z 315.013,A -85,B 0,C 180,E1 -22026.381,E2 -22026.381} C_VEL
LIN {X 0,Y 189.035,Z 327.628,A -85,B 0,C 180,E1 -22028.433,E2 -22028.433} C_VEL
LIN {X 0,Y 187.341,Z 339.147,A -85,B 0,C 180,E1 -22030.838,E2 -22030.838} C_VEL
LIN {X 0,Y 185.946,Z 349.292,A -85,B 0,C 180,E1 -22033.534,E2 -22033.534} C_VEL
LIN {X 0,Y 184.949,Z 357.603,A -85,B 0,C 180,E1 -22036.262,E2 -22036.262} C_VEL
LIN {X 0,Y 184.131,Z 365.715,A -85,B 0,C 180,E1 -22039.555,E2 -22039.555} C_VEL
LIN {X 0,Y 183.869,Z 371.178,A -85,B 0,C 180,E1 -22042.313,E2 -22042.313} C_VEL
LIN {X 0,Y 183.797,Z 376.434,A -85,B 0,C 180,E1 -22045.615,E2 -22045.615} C_VEL
LIN {X 0,Y 183.808,Z 380.388,A -85,B 0,C 180,E1 -22048.905,E2 -22048.905} C_VEL
LIN {X 0,Y 183.902,Z 381.432,A -85,B 0,C 180,E1 -22050.001,E2 -22050.001} C_VEL
LIN {X 0,Y 183.528,Z 383.147,A -85,B 0,C 180,E1 -22052.195,E2 -22052.195} C_VEL
LIN {X 0,Y 183.333,Z 384.527,A -85,B 0,C 180,E1 -22054.645,E2 -22054.645} C_VEL
LIN {X 0,Y 183.47,Z 385.707,A -85,B 0,C 180,E1 -22058.815,E2 -22058.815} C_VEL
LIN {X 0,Y 184.568,Z 385.501,A -85,B 0,C 180,E1 -22063.208,E2 -22063.208} C_VEL
LIN {X 0,Y 185.489,Z 384.825,A -85,B 0,C 180,E1 -22065.381,E2 -22065.381} C_VEL
LIN {X 0,Y 188.447,Z 382.321,A -85,B 0,C 180,E1 -22069.613,E2 -22069.613} C_VEL
LIN {X 0,Y 192.368,Z 378.287,A -85,B 0,C 180,E1 -22073.696,E2 -22073.696} C_VEL
LIN {X 0,Y 196.029,Z 374.112,A -85,B 0,C 180,E1 -22076.626,E2 -22076.626} C_VEL
LIN {X 0,Y 200.427,Z 368.926,A -85,B 0,C 180,E1 -22079.401,E2 -22079.401} C_VEL
LIN {X 0,Y 206.125,Z 361.368,A -85,B 0,C 180,E1 -22082.481,E2 -22082.481} C_VEL
LIN {X 0,Y 212.729,Z 351.796,A -85,B 0,C 180,E1 -22085.321,E2 -22085.321} C_VEL
LIN {X 0,Y 218.874,Z 341.665,A -85,B 0,C 180,E1 -22087.596,E2 -22087.596} C_VEL
LIN {X 0,Y 224.286,Z 331.371,A -85,B 0,C 180,E1 -22089.386,E2 -22089.386} C_VEL
LIN {X 0,Y 229.589,Z 319.924,A -85,B 0,C 180,E1 -22090.868,E2 -22090.868} C_VEL
LIN {X 0,Y 234.46,Z 307.22,A -85,B 0,C 180,E1 -22092.122,E2 -22092.122} C_VEL
LIN {X 0,Y 238.577,Z 293.98,A -85,B 0,C 180,E1 -22093.079,E2 -22093.079} C_VEL
LIN {X 0,Y 241.716,Z 280.253,A -85,B 0,C 180,E1 -22093.796,E2 -22093.796} C_VEL
LIN {X 0,Y 246.195,Z 249.524,A -85,B 0,C 180,E1 -22095.045,E2 -22095.045} C_VEL
LIN {X 0,Y 244.631,Z 243.989,A -85,B 0,C 180,E1 -22096.78,E2 -22096.78} C_VEL
LIN {X 0,Y 242.907,Z 238.435,A -85,B 0,C 180,E1 -22098.973,E2 -22098.973} C_VEL
LIN {X 0,Y 241.346,Z 233.892,A -85,B 0,C 180,E1 -22101.54,E2 -22101.54} C_VEL
LIN {X 0,Y 240.019,Z 229.239,A -85,B 0,C 180,E1 -22105.775,E2 -22105.775} C_VEL
LIN {X 0,Y 239.839,Z 228.361,A -85,B 0,C 180,E1 -22108.166,E2 -22108.166} C_VEL
LIN {X 0,Y 240.278,Z 228.518,A -85,B 0,C 180,E1 -22110.795,E2 -22110.795} C_VEL
LIN {X 0,Y 241.929,Z 230.569,A -85,B 0,C 180,E1 -22114.483,E2 -22114.483} C_VEL
LIN {X 0,Y 243.698,Z 233.615,A -85,B 0,C 180,E1 -22116.973,E2 -22116.973} C_VEL
LIN {X 0,Y 245.502,Z 237.027,A -85,B 0,C 180,E1 -22118.931,E2 -22118.931} C_VEL
LIN {X 0,Y 247.153,Z 240.758,A -85,B 0,C 180,E1 -22120.559,E2 -22120.559} C_VEL
LIN {X 0,Y 242.686,Z 270.843,A -85,B 0,C 180,E1 -22121.758,E2 -22121.758} C_VEL
LIN {X 0,Y 240.116,Z 282.968,A -85,B 0,C 180,E1 -22122.49,E2 -22122.49} C_VEL
LIN {X 0,Y 236.869,Z 294.626,A -85,B 0,C 180,E1 -22123.447,E2 -22123.447} C_VEL
LIN {X 0,Y 232.615,Z 306.679,A -85,B 0,C 180,E1 -22124.757,E2 -22124.757} C_VEL
LIN {X 0,Y 227.652,Z 318.296,A -85,B 0,C 180,E1 -22126.384,E2 -22126.384} C_VEL
LIN {X 0,Y 222.592,Z 328.239,A -85,B 0,C 180,E1 -22128.177,E2 -22128.177} C_VEL
LIN {X 0,Y 217.379,Z 337.062,A -85,B 0,C 180,E1 -22130.227,E2 -22130.227} C_VEL
LIN {X 0,Y 211.482,Z 345.787,A -85,B 0,C 180,E1 -22132.84,E2 -22132.84} C_VEL
LIN {X 0,Y 206.062,Z 352.745,A -85,B 0,C 180,E1 -22135.598,E2 -22135.598} C_VEL
LIN {X 0,Y 200.422,Z 359.004,A -85,B 0,C 180,E1 -22138.995,E2 -22138.995} C_VEL
LIN {X 0,Y 196.176,Z 363.025,A -85,B 0,C 180,E1 -22142.052,E2 -22142.052} C_VEL
LIN {X 0,Y 193.686,Z 365.052,A -85,B 0,C 180,E1 -22144.161,E2 -22144.161} C_VEL
LIN {X 0,Y 191.072,Z 366.849,A -85,B 0,C 180,E1 -22146.723,E2 -22146.723} C_VEL
LIN {X 0,Y 187.838,Z 368.315,A -85,B 0,C 180,E1 -22150.781,E2 -22150.781} C_VEL
LIN {X 0,Y 186.406,Z 368.488,A -85,B 0,C 180,E1 -22153.074,E2 -22153.074} C_VEL
LIN {X 0,Y 185.241,Z 368.23,A -85,B 0,C 180,E1 -22155.4,E2 -22155.4} C_VEL
LIN {X 0,Y 184.329,Z 367.475,A -85,B 0,C 180,E1 -22157.758,E2 -22157.758} C_VEL
LIN {X 0,Y 183.67,Z 366.247,A -85,B 0,C 180,E1 -22160.143,E2 -22160.143} C_VEL
LIN {X 0,Y 183.191,Z 364.195,A -85,B 0,C 180,E1 -22162.963,E2 -22162.963} C_VEL
LIN {X 0,Y 183.082,Z 360.983,A -85,B 0,C 180,E1 -22166.196,E2 -22166.196} C_VEL
LIN {X 0,Y 183.399,Z 356.018,A -85,B 0,C 180,E1 -22169.878,E2 -22169.878} C_VEL
LIN {X 0,Y 183.905,Z 351.05,A -85,B 0,C 180,E1 -22172.781,E2 -22172.781} C_VEL
LIN {X 0,Y 184.646,Z 344.296,A -85,B 0,C 180,E1 -22175.968,E2 -22175.968} C_VEL
LIN {X 0,Y 185.758,Z 335.441,A -85,B 0,C 180,E1 -22179.324,E2 -22179.324} C_VEL
LIN {X 0,Y 187.091,Z 326.277,A -85,B 0,C 180,E1 -22182.103,E2 -22182.103} C_VEL
LIN {X 0,Y 188.585,Z 315.265,A -85,B 0,C 180,E1 -22184.795,E2 -22184.795} C_VEL
LIN {X 0,Y 190.086,Z 304.502,A -85,B 0,C 180,E1 -22186.903,E2 -22186.903} C_VEL
LIN {X 0,Y 191.605,Z 291.866,A -85,B 0,C 180,E1 -22188.841,E2 -22188.841} C_VEL
LIN {X 0,Y 192.932,Z 279.317,A -85,B 0,C 180,E1 -22190.31,E2 -22190.31} C_VEL
LIN {X 0,Y 193.918,Z 264.944,A -85,B 0,C 180,E1 -22191.498,E2 -22191.498} C_VEL
LIN {X 0,Y 197.564,Z 199.943,A -85,B 0,C 180,E1 -22194.762,E2 -22194.762} C_VEL
LIN {X 0,Y 197.175,Z 197.68,A -85,B 0,C 180,E1 -22194.917,E2 -22194.917} C_VEL
LIN {X 0,Y 186.14,Z 167.283,A -85,B 0,C 180,E1 -22197.639,E2 -22197.639} C_VEL
LIN {X 0,Y 185.644,Z 165.362,A -85,B 0,C 180,E1 -22197.881,E2 -22197.881} C_VEL
LIN {X 0,Y 185.562,Z 165.374,A -85,B 0,C 180,E1 -22202.967,E2 -22202.967} C_VEL
LIN {X 0,Y 185.59,Z 165.367,A -85,B 0,C 180,E1 -22207.747,E2 -22207.747} C_VEL
LIN {X 0,Y 185.657,Z 165.357,A -85,B 0,C 180,E1 -22212.371,E2 -22212.371} C_VEL
LIN {X 0,Y 185.724,Z 165.347,A -85,B 0,C 180,E1 -22216.876,E2 -22216.876} C_VEL
LIN {X 0,Y 186.008,Z 165.315,A -85,B 0,C 180,E1 -22221.307,E2 -22221.307} C_VEL
LIN {X 0,Y 186.207,Z 165.289,A -85,B 0,C 180,E1 -22227.836,E2 -22227.836} C_VEL
LIN {X 0,Y 186.406,Z 165.264,A -85,B 0,C 180,E1 -22229.999,E2 -22229.999} C_VEL
LIN {X 0,Y 185.923,Z 165.322,A -85,B 0,C 180,E1 -22234.335,E2 -22234.335} C_VEL
LIN {X 0,Y 186.007,Z 165.315,A -85,B 0,C 180,E1 -22238.692,E2 -22238.692} C_VEL
LIN {X 0,Y 185.762,Z 165.344,A -85,B 0,C 180,E1 -22243.12,E2 -22243.12} C_VEL
LIN {X 0,Y 185.672,Z 165.352,A -85,B 0,C 180,E1 -22248.866,E2 -22248.866} C_VEL
LIN {X 0,Y 185.574,Z 165.368,A -85,B 0,C 180,E1 -22254.646,E2 -22254.646} C_VEL
LIN {X 0,Y 185.576,Z 165.365,A -85,B 0,C 180,E1 -22259.493,E2 -22259.493} C_VEL
LIN {X 0,Y 185.518,Z 165.373,A -85,B 0,C 180,E1 -22264.627,E2 -22264.627} C_VEL
LIN {X 0,Y 185.565,Z 165.366,A -85,B 0,C 180,E1 -22267.314,E2 -22267.314} C_VEL
LIN {X 0,Y 185.559,Z 165.37,A -85,B 0,C 180,E1 -22270.757,E2 -22270.757} C_VEL
LIN {X 0,Y 185.561,Z 165.37,A -85,B 0,C 180,E1 -22276.021,E2 -22276.021} C_VEL
LIN {X 0,Y 185.537,Z 165.373,A -85,B 0,C 180,E1 -22279.914,E2 -22279.914} C_VEL
LIN {X 0,Y 185.556,Z 165.365,A -85,B 0,C 180,E1 -22282.7,E2 -22282.7} C_VEL
LIN {X 0,Y 185.543,Z 165.372,A -85,B 0,C 180,E1 -22287.976,E2 -22287.976} C_VEL
LIN {X 0,Y 185.579,Z 165.363,A -85,B 0,C 180,E1 -22290.576,E2 -22290.576} C_VEL
LIN {X 0,Y 185.585,Z 165.369,A -85,B 0,C 180,E1 -22295.383,E2 -22295.383} C_VEL
LIN {X 0,Y 185.672,Z 165.355,A -85,B 0,C 180,E1 -22301.134,E2 -22301.134} C_VEL
LIN {X 0,Y 185.722,Z 165.35,A -85,B 0,C 180,E1 -22304.64,E2 -22304.64} C_VEL
LIN {X 0,Y 185.922,Z 165.326,A -85,B 0,C 180,E1 -22309.36,E2 -22309.36} C_VEL
LIN {X 0,Y 185.959,Z 165.319,A -85,B 0,C 180,E1 -22313.491,E2 -22313.491} C_VEL
LIN {X 0,Y 186.206,Z 165.288,A -85,B 0,C 180,E1 -22317.838,E2 -22317.838} C_VEL
